SPLINE
SPL {X  -111.648, Y  +797.871, Z    +0.000, E1   -60.847, E3 +126698.241}
SPL {X  -149.288, Y  +747.285, Z    +0.000, E1   -46.770, E3 +126694.232}
SPL {X  -159.627, Y  +719.761, Z    +0.000, E1   -35.247, E3 +126699.297}
SPL {X  -164.185, Y  +697.485, Z    +0.000, E1   -20.950, E3 +126699.616}
SPL {X  -165.453, Y  +683.578, Z    +0.000, E1    -9.445, E3 +126698.203}
SPL {X  -165.642, Y  +677.105, Z    +0.000, E1    -3.559, E3 +126698.514}
SPL {X  -165.650, Y  +673.522, Z    +0.000, E1    -0.038, E3 +126697.362}
SPL {X  -165.650, Y  +671.354, Z    +0.000, E1    +3.728, E3 +126696.849}
SPL {X  -165.650, Y  +666.485, Z    +0.000, E1   +14.169, E3 +126696.576}
SPL {X  -165.650, Y  +661.236, Z    +0.000, E1   +26.072, E3 +126696.266}
SPL {X  -165.650, Y  +655.357, Z    +0.000, E1   +38.693, E3 +126695.493}
SPL {X  -165.650, Y  +646.637, Z    +0.000, E1   +52.169, E3 +126695.275}
SPL {X  -165.650, Y  +637.909, Z    +0.000, E1   +64.161, E3 +126692.070}
SPL {X  -165.650, Y  +618.963, Z    +0.000, E1   +72.815, E3 +126693.133}
SPL {X  -165.650, Y  +575.208, Z    +0.000, E1   +76.222, E3 +126704.394}
SPL {X  -165.650, Y  +394.754, Z    +0.000, E1   +73.248, E3 +126799.541}
ENDSPLINE

SPLINE
SPL {X  -165.650, Y  +407.500, Z    +0.000, E1   +70.919, E3 +126814.162}
ENDSPLINE

SPLINE
SPL {X  -165.650, Y  +384.687, Z    +0.000, E1   +71.028, E3 +126829.408}
SPL {X  -164.996, Y  +363.797, Z    +0.000, E1   +70.987, E3 +126844.383}
SPL {X  -162.841, Y  +348.123, Z    +0.000, E1   +70.683, E3 +126858.311}
SPL {X  -162.352, Y  +345.609, Z    +0.000, E1   +69.290, E3 +126872.264}
SPL {X  -157.663, Y  +327.685, Z    +0.000, E1   +69.808, E3 +126881.124}
SPL {X  -152.892, Y  +314.750, Z    +0.000, E1   +69.675, E3 +126891.339}
SPL {X  -149.246, Y  +306.628, Z    +0.000, E1   +69.029, E3 +126901.808}
SPL {X  -145.495, Y  +299.310, Z    +0.000, E1   +68.659, E3 +126909.416}
SPL {X  -142.111, Y  +293.387, Z    +0.000, E1   +68.421, E3 +126915.058}
SPL {X  -138.525, Y  +287.667, Z    +0.000, E1   +67.662, E3 +126923.618}
SPL {X  -134.450, Y  +281.737, Z    +0.000, E1   +67.268, E3 +126929.723}
SPL {X  -131.812, Y  +278.173, Z    +0.000, E1   +66.669, E3 +126935.071}
SPL {X  -128.148, Y  +273.533, Z    +0.000, E1   +67.328, E3 +126935.430}
SPL {X  -116.216, Y  +260.459, Z    +0.000, E1   +70.200, E3 +126931.736}
SPL {X   -66.125, Y  +226.621, Z    +0.000, E1   +55.862, E3 +127094.634}
ENDSPLINE

SPLINE
SPL {X  -111.531, Y  +256.023, Z    +0.000, E1   +58.853, E3 +127237.516}
SPL {X  -139.240, Y  +288.767, Z    +0.000, E1   +52.898, E3 +127247.689}
SPL {X  -156.827, Y  +325.161, Z    +0.000, E1   +39.042, E3 +127246.059}
SPL {X  -162.324, Y  +345.471, Z    +0.000, E1   +27.849, E3 +127246.527}
SPL {X  -164.696, Y  +360.744, Z    +0.000, E1   +17.229, E3 +127247.441}
SPL {X  -165.561, Y  +373.081, Z    +0.000, E1    +6.973, E3 +127246.185}
SPL {X  -165.650, Y  +379.105, Z    +0.000, E1    +1.379, E3 +127245.746}
SPL {X  -165.650, Y  +380.899, Z    +0.000, E1    -0.394, E3 +127244.884}
SPL {X  -165.650, Y  +385.044, Z    +0.000, E1    -8.496, E3 +127244.300}
SPL {X  -165.650, Y  +388.717, Z    +0.000, E1   -16.400, E3 +127244.156}
SPL {X  -165.650, Y  +394.613, Z    +0.000, E1   -29.184, E3 +127243.625}
SPL {X  -165.650, Y  +402.836, Z    +0.000, E1   -44.797, E3 +127243.027}
SPL {X  -165.650, Y  +416.111, Z    +0.000, E1   -60.729, E3 +127242.094}
SPL {X  -165.650, Y  +457.077, Z    +0.000, E1   -75.210, E3 +127245.418}
SPL {X  -165.650, Y  +475.293, Z    +0.000, E1   -75.741, E3 +127251.195}
SPL {X  -164.204, Y  +697.342, Z    +0.000, E1   -76.015, E3 +127338.170}
ENDSPLINE

SPLINE
SPL {X  -165.650, Y  +664.340, Z    +0.000, E1   -71.862, E3 +127363.574}
ENDSPLINE

SPLINE
SPL {X  -165.237, Y  +687.187, Z    +0.000, E1   -71.947, E3 +127377.835}
SPL {X  -163.865, Y  +699.752, Z    +0.000, E1   -71.643, E3 +127389.241}
SPL {X  -161.821, Y  +710.908, Z    +0.000, E1   -71.322, E3 +127399.781}
SPL {X  -158.993, Y  +721.987, Z    +0.000, E1   -71.173, E3 +127408.569}
SPL {X  -155.811, Y  +731.738, Z    +0.000, E1   -70.890, E3 +127417.577}
SPL {X  -152.643, Y  +739.844, Z    +0.000, E1   -70.463, E3 +127426.436}
SPL {X  -149.782, Y  +746.247, Z    +0.000, E1   -70.149, E3 +127433.126}
SPL {X  -146.450, Y  +752.910, Z    +0.000, E1   -69.680, E3 +127441.004}
SPL {X  -143.017, Y  +759.082, Z    +0.000, E1   -69.156, E3 +127448.615}
SPL {X  -140.057, Y  +763.953, Z    +0.000, E1   -68.829, E3 +127453.855}
SPL {X  -136.535, Y  +769.298, Z    +0.000, E1   -68.442, E3 +127459.716}
SPL {X  -133.553, Y  +773.498, Z    +0.000, E1   -67.773, E3 +127465.881}
SPL {X  -129.830, Y  +778.379, Z    +0.000, E1   -67.491, E3 +127470.507}
SPL {X  -116.788, Y  +792.975, Z    +0.000, E1   -71.297, E3 +127463.891}
SPL {X   -64.927, Y  +827.895, Z    +0.000, E1   -57.691, E3 +127589.494}
ENDSPLINE

SPLINE
SPL {X  -111.648, Y  +797.871, Z    +0.000, E1   -60.847, E3 +127786.477}
SPL {X  -149.288, Y  +747.285, Z    +0.000, E1   -46.770, E3 +127782.468}
SPL {X  -159.627, Y  +719.761, Z    +0.000, E1   -35.247, E3 +127787.533}
SPL {X  -164.185, Y  +697.485, Z    +0.000, E1   -20.950, E3 +127787.852}
SPL {X  -165.594, Y  +679.817, Z    +0.000, E1    -6.204, E3 +127786.628}
SPL {X  -165.650, Y  +673.522, Z    +0.000, E1    -0.038, E3 +127785.597}
SPL {X  -165.650, Y  +671.354, Z    +0.000, E1    +3.728, E3 +127785.085}
SPL {X  -165.650, Y  +666.485, Z    +0.000, E1   +14.169, E3 +127784.812}
SPL {X  -165.650, Y  +661.236, Z    +0.000, E1   +26.072, E3 +127784.501}
SPL {X  -165.650, Y  +655.357, Z    +0.000, E1   +38.693, E3 +127783.728}
SPL {X  -165.650, Y  +646.637, Z    +0.000, E1   +52.169, E3 +127783.510}
SPL {X  -165.650, Y  +637.909, Z    +0.000, E1   +64.161, E3 +127780.306}
SPL {X  -165.650, Y  +618.963, Z    +0.000, E1   +72.815, E3 +127781.369}
SPL {X  -165.650, Y  +575.208, Z    +0.000, E1   +76.222, E3 +127792.629}
SPL {X  -165.650, Y  +394.754, Z    +0.000, E1   +73.248, E3 +127887.776}
ENDSPLINE

SPLINE
SPL {X  -165.650, Y  +407.500, Z    +0.000, E1   +70.919, E3 +127902.397}
ENDSPLINE

SPLINE
SPL {X  -165.650, Y  +390.855, Z    +0.000, E1   +71.004, E3 +127913.325}
SPL {X  -165.534, Y  +372.295, Z    +0.000, E1   +71.066, E3 +127925.875}
SPL {X  -164.039, Y  +355.451, Z    +0.000, E1   +70.703, E3 +127941.273}
SPL {X  -161.297, Y  +340.777, Z    +0.000, E1   +70.794, E3 +127950.566}
ENDSPLINE

SPLINE
SPL {X  -162.352, Y  +345.609, Z    +0.000, E1   +69.290, E3 +127960.499}
ENDSPLINE

SPLINE
SPL {X  -159.253, Y  +332.909, Z    +0.000, E1   +69.652, E3 +127966.845}
SPL {X  -155.267, Y  +320.775, Z    +0.000, E1   +69.854, E3 +127973.939}
SPL {X  -151.256, Y  +310.961, Z    +0.000, E1   +69.467, E3 +127983.814}
SPL {X  -148.628, Y  +305.359, Z    +0.000, E1   +68.848, E3 +127992.092}
SPL {X  -145.495, Y  +299.310, Z    +0.000, E1   +68.659, E3 +127997.651}
SPL {X  -142.111, Y  +293.387, Z    +0.000, E1   +68.421, E3 +128003.293}
SPL {X  -138.525, Y  +287.667, Z    +0.000, E1   +67.662, E3 +128011.853}
SPL {X  -134.450, Y  +281.737, Z    +0.000, E1   +67.268, E3 +128017.958}
SPL {X  -131.812, Y  +278.173, Z    +0.000, E1   +66.669, E3 +128023.307}
SPL {X  -128.148, Y  +273.533, Z    +0.000, E1   +67.328, E3 +128023.665}
SPL {X  -116.216, Y  +260.459, Z    +0.000, E1   +70.200, E3 +128019.972}
SPL {X   -66.125, Y  +226.621, Z    +0.000, E1   +55.862, E3 +128182.870}
ENDSPLINE

SPLINE
SPL {X  -111.531, Y  +256.023, Z    +0.000, E1   +58.853, E3 +128325.752}
SPL {X  -139.240, Y  +288.767, Z    +0.000, E1   +52.898, E3 +128335.925}
SPL {X  -156.827, Y  +325.161, Z    +0.000, E1   +39.042, E3 +128334.294}
SPL {X  -163.133, Y  +349.734, Z    +0.000, E1   +25.193, E3 +128335.419}
SPL {X  -165.214, Y  +366.494, Z    +0.000, E1   +12.605, E3 +128334.891}
SPL {X  -165.615, Y  +375.073, Z    +0.000, E1    +5.133, E3 +128334.379}
SPL {X  -165.650, Y  +380.392, Z    +0.000, E1    +0.180, E3 +128333.338}
SPL {X  -165.650, Y  +381.828, Z    +0.000, E1    -2.219, E3 +128332.736}
SPL {X  -165.650, Y  +385.044, Z    +0.000, E1    -8.496, E3 +128332.535}
SPL {X  -165.650, Y  +388.717, Z    +0.000, E1   -16.400, E3 +128332.391}
SPL {X  -165.650, Y  +394.613, Z    +0.000, E1   -29.184, E3 +128331.860}
SPL {X  -165.650, Y  +402.836, Z    +0.000, E1   -44.797, E3 +128331.263}
SPL {X  -165.650, Y  +416.111, Z    +0.000, E1   -60.729, E3 +128330.329}
SPL {X  -165.650, Y  +471.994, Z    +0.000, E1   -75.670, E3 +128338.383}
SPL {X  -164.204, Y  +697.342, Z    +0.000, E1   -76.015, E3 +128426.405}
ENDSPLINE

SPLINE
SPL {X  -165.650, Y  +664.340, Z    +0.000, E1   -71.862, E3 +128451.809}
ENDSPLINE

SPLINE
SPL {X  -165.237, Y  +687.187, Z    +0.000, E1   -71.947, E3 +128466.070}
SPL {X  -163.865, Y  +699.752, Z    +0.000, E1   -71.643, E3 +128477.476}
SPL {X  -161.821, Y  +710.908, Z    +0.000, E1   -71.322, E3 +128488.016}
SPL {X  -158.993, Y  +721.987, Z    +0.000, E1   -71.173, E3 +128496.804}
SPL {X  -155.811, Y  +731.738, Z    +0.000, E1   -70.890, E3 +128505.812}
SPL {X  -152.643, Y  +739.844, Z    +0.000, E1   -70.463, E3 +128514.672}
SPL {X  -149.782, Y  +746.247, Z    +0.000, E1   -70.149, E3 +128521.361}
SPL {X  -146.450, Y  +752.910, Z    +0.000, E1   -69.680, E3 +128529.239}
SPL {X  -143.017, Y  +759.082, Z    +0.000, E1   -69.156, E3 +128536.851}
SPL {X  -140.057, Y  +763.953, Z    +0.000, E1   -68.829, E3 +128542.090}
SPL {X  -136.535, Y  +769.298, Z    +0.000, E1   -68.442, E3 +128547.952}
SPL {X  -132.359, Y  +775.105, Z    +0.000, E1   -67.661, E3 +128555.809}
SPL {X  -128.720, Y  +779.765, Z    +0.000, E1   -67.454, E3 +128559.790}
SPL {X  -116.788, Y  +792.975, Z    +0.000, E1   -71.297, E3 +128552.127}
SPL {X   -70.520, Y  +825.390, Z    +0.000, E1   -59.928, E3 +128646.037}
SPL {X   -62.607, Y  +828.863, Z    +0.000, E1   -56.584, E3 +128700.922}
ENDSPLINE

SPLINE
SPL {X  -111.648, Y  +797.871, Z    +0.000, E1   -60.847, E3 +128874.712}
SPL {X  -149.288, Y  +747.285, Z    +0.000, E1   -46.770, E3 +128870.703}
SPL {X  -161.496, Y  +712.364, Z    +0.000, E1   -31.137, E3 +128876.498}
SPL {X  -164.701, Y  +693.202, Z    +0.000, E1   -17.512, E3 +128875.472}
SPL {X  -165.594, Y  +679.817, Z    +0.000, E1    -6.204, E3 +128874.863}
SPL {X  -165.650, Y  +673.263, Z    +0.000, E1    +0.216, E3 +128873.745}
SPL {X  -165.650, Y  +670.095, Z    +0.000, E1    +6.482, E3 +128873.148}
SPL {X  -165.650, Y  +666.485, Z    +0.000, E1   +14.169, E3 +128873.047}
SPL {X  -165.650, Y  +661.236, Z    +0.000, E1   +26.072, E3 +128872.736}
SPL {X  -165.650, Y  +655.357, Z    +0.000, E1   +38.693, E3 +128871.964}
SPL {X  -165.650, Y  +646.637, Z    +0.000, E1   +52.169, E3 +128871.745}
SPL {X  -165.650, Y  +637.909, Z    +0.000, E1   +64.161, E3 +128868.541}
SPL {X  -165.650, Y  +618.963, Z    +0.000, E1   +72.815, E3 +128869.604}
SPL {X  -165.650, Y  +575.208, Z    +0.000, E1   +76.222, E3 +128880.865}
SPL {X  -165.650, Y  +394.754, Z    +0.000, E1   +73.248, E3 +128976.011}
ENDSPLINE

SPLINE
SPL {X  -165.650, Y  +407.500, Z    +0.000, E1   +70.919, E3 +128990.632}
ENDSPLINE

SPLINE
SPL {X  -165.650, Y  +390.855, Z    +0.000, E1   +71.004, E3 +129001.560}
SPL {X  -165.534, Y  +372.295, Z    +0.000, E1   +71.066, E3 +129014.110}
SPL {X  -164.039, Y  +355.451, Z    +0.000, E1   +70.703, E3 +129029.509}
SPL {X  -161.297, Y  +340.777, Z    +0.000, E1   +70.794, E3 +129038.801}
ENDSPLINE

SPLINE
SPL {X  -162.352, Y  +345.609, Z    +0.000, E1   +69.290, E3 +129048.734}
ENDSPLINE

SPLINE
SPL {X  -157.663, Y  +327.685, Z    +0.000, E1   +69.808, E3 +129057.594}
SPL {X  -152.892, Y  +314.750, Z    +0.000, E1   +69.675, E3 +129067.810}
SPL {X  -149.246, Y  +306.628, Z    +0.000, E1   +69.029, E3 +129078.278}
SPL {X  -145.495, Y  +299.310, Z    +0.000, E1   +68.659, E3 +129085.887}
SPL {X  -142.111, Y  +293.387, Z    +0.000, E1   +68.421, E3 +129091.528}
SPL {X  -138.525, Y  +287.667, Z    +0.000, E1   +67.662, E3 +129100.088}
SPL {X  -134.450, Y  +281.737, Z    +0.000, E1   +67.268, E3 +129106.193}
SPL {X  -131.812, Y  +278.173, Z    +0.000, E1   +66.669, E3 +129111.542}
SPL {X  -128.148, Y  +273.533, Z    +0.000, E1   +67.328, E3 +129111.900}
SPL {X  -116.216, Y  +260.459, Z    +0.000, E1   +70.200, E3 +129108.207}
SPL {X   -66.125, Y  +226.621, Z    +0.000, E1   +55.862, E3 +129271.105}
ENDSPLINE

SPLINE
SPL {X  -111.531, Y  +256.023, Z    +0.000, E1   +58.853, E3 +129413.987}
SPL {X  -139.240, Y  +288.767, Z    +0.000, E1   +52.898, E3 +129424.160}
SPL {X  -156.827, Y  +325.161, Z    +0.000, E1   +39.042, E3 +129422.529}
SPL {X  -162.324, Y  +345.471, Z    +0.000, E1   +27.849, E3 +129422.998}
SPL {X  -165.055, Y  +364.477, Z    +0.000, E1   +14.326, E3 +129423.436}
SPL {X  -165.646, Y  +377.353, Z    +0.000, E1    +3.112, E3 +129422.393}
SPL {X  -165.650, Y  +380.500, Z    +0.000, E1    -0.000, E3 +129421.519}
SPL {X  -165.650, Y  +381.828, Z    +0.000, E1    -2.219, E3 +129420.971}
SPL {X  -165.650, Y  +385.044, Z    +0.000, E1    -8.496, E3 +129420.771}
SPL {X  -165.650, Y  +390.492, Z    +0.000, E1   -20.084, E3 +129420.425}
SPL {X  -165.650, Y  +400.081, Z    +0.000, E1   -39.836, E3 +129419.730}
SPL {X  -165.650, Y  +416.111, Z    +0.000, E1   -60.729, E3 +129418.565}
SPL {X  -165.650, Y  +471.994, Z    +0.000, E1   -75.670, E3 +129426.618}
SPL {X  -164.204, Y  +697.342, Z    +0.000, E1   -76.015, E3 +129514.641}
ENDSPLINE

SPLINE
SPL {X  -165.650, Y  +656.030, Z    +0.000, E1   -71.686, E3 +129536.080}
ENDSPLINE

SPLINE
SPL {X  -165.610, Y  +679.119, Z    +0.000, E1   -71.889, E3 +129549.703}
SPL {X  -163.827, Y  +700.009, Z    +0.000, E1   -71.824, E3 +129564.269}
SPL {X  -161.041, Y  +714.304, Z    +0.000, E1   -71.423, E3 +129577.615}
SPL {X  -159.124, Y  +721.538, Z    +0.000, E1   -70.872, E3 +129587.267}
SPL {X  -155.811, Y  +731.738, Z    +0.000, E1   -70.890, E3 +129594.048}
SPL {X  -152.643, Y  +739.844, Z    +0.000, E1   -70.463, E3 +129602.907}
SPL {X  -149.782, Y  +746.247, Z    +0.000, E1   -70.149, E3 +129609.597}
SPL {X  -146.450, Y  +752.910, Z    +0.000, E1   -69.680, E3 +129617.475}
SPL {X  -143.017, Y  +759.082, Z    +0.000, E1   -69.156, E3 +129625.086}
SPL {X  -139.030, Y  +765.558, Z    +0.000, E1   -68.719, E3 +129632.119}
SPL {X  -135.682, Y  +770.527, Z    +0.000, E1   -68.337, E3 +129637.503}
SPL {X  -133.553, Y  +773.498, Z    +0.000, E1   -67.773, E3 +129642.352}
SPL {X  -129.830, Y  +778.379, Z    +0.000, E1   -67.491, E3 +129646.978}
SPL {X  -116.788, Y  +792.975, Z    +0.000, E1   -71.297, E3 +129640.362}
SPL {X   -70.520, Y  +825.390, Z    +0.000, E1   -59.928, E3 +129734.272}
SPL {X   -62.607, Y  +828.863, Z    +0.000, E1   -56.584, E3 +129789.157}
ENDSPLINE

SPLINE
SPL {X  -111.648, Y  +797.871, Z    +0.000, E1   -60.847, E3 +129962.947}
SPL {X  -149.288, Y  +747.285, Z    +0.000, E1   -46.770, E3 +129958.938}
SPL {X  -161.496, Y  +712.364, Z    +0.000, E1   -31.137, E3 +129964.733}
SPL {X  -164.701, Y  +693.202, Z    +0.000, E1   -17.512, E3 +129963.708}
SPL {X  -165.453, Y  +683.578, Z    +0.000, E1    -9.445, E3 +129962.909}
SPL {X  -165.642, Y  +677.105, Z    +0.000, E1    -3.559, E3 +129963.220}
SPL {X  -165.650, Y  +673.263, Z    +0.000, E1    +0.216, E3 +129961.980}
SPL {X  -165.650, Y  +670.095, Z    +0.000, E1    +6.482, E3 +129961.384}
SPL {X  -165.650, Y  +666.485, Z    +0.000, E1   +14.169, E3 +129961.282}
SPL {X  -165.650, Y  +661.236, Z    +0.000, E1   +26.072, E3 +129960.971}
SPL {X  -165.650, Y  +653.063, Z    +0.000, E1   +42.395, E3 +129960.375}
SPL {X  -165.650, Y  +640.535, Z    +0.000, E1   +60.776, E3 +129957.860}
SPL {X  -165.650, Y  +618.963, Z    +0.000, E1   +72.815, E3 +129957.839}
SPL {X  -165.650, Y  +575.208, Z    +0.000, E1   +76.222, E3 +129969.100}
SPL {X  -165.650, Y  +394.754, Z    +0.000, E1   +73.248, E3 +130064.246}
ENDSPLINE

SPLINE
SPL {X  -165.650, Y  +407.500, Z    +0.000, E1   +70.919, E3 +130078.868}
ENDSPLINE

SPLINE
SPL {X  -165.650, Y  +384.687, Z    +0.000, E1   +71.028, E3 +130094.114}
SPL {X  -164.996, Y  +363.797, Z    +0.000, E1   +70.987, E3 +130109.089}
SPL {X  -162.841, Y  +348.123, Z    +0.000, E1   +70.683, E3 +130123.016}
SPL {X  -162.352, Y  +345.609, Z    +0.000, E1   +69.290, E3 +130136.969}
SPL {X  -159.253, Y  +332.909, Z    +0.000, E1   +69.652, E3 +130143.316}
SPL {X  -156.309, Y  +323.661, Z    +0.000, E1   +69.908, E3 +130147.831}
SPL {X  -152.892, Y  +314.750, Z    +0.000, E1   +69.675, E3 +130156.045}
SPL {X  -149.246, Y  +306.628, Z    +0.000, E1   +69.029, E3 +130166.513}
SPL {X  -144.614, Y  +297.712, Z    +0.000, E1   +68.717, E3 +130174.867}
SPL {X  -141.011, Y  +291.576, Z    +0.000, E1   +68.040, E3 +130183.345}
SPL {X  -137.649, Y  +286.345, Z    +0.000, E1   +67.498, E3 +130190.039}
SPL {X  -134.450, Y  +281.737, Z    +0.000, E1   +67.268, E3 +130194.429}
SPL {X  -131.812, Y  +278.173, Z    +0.000, E1   +66.669, E3 +130199.777}
SPL {X  -128.148, Y  +273.533, Z    +0.000, E1   +67.328, E3 +130200.136}
SPL {X  -116.216, Y  +260.459, Z    +0.000, E1   +70.200, E3 +130196.442}
SPL {X   -66.125, Y  +226.621, Z    +0.000, E1   +55.862, E3 +130359.340}
ENDSPLINE

SPLINE
SPL {X  -111.531, Y  +256.023, Z    +0.000, E1   +58.853, E3 +130502.222}
SPL {X  -139.240, Y  +288.767, Z    +0.000, E1   +52.898, E3 +130512.395}
SPL {X  -156.827, Y  +325.161, Z    +0.000, E1   +39.042, E3 +130510.764}
SPL {X  -162.324, Y  +345.471, Z    +0.000, E1   +27.849, E3 +130511.233}
SPL {X  -164.696, Y  +360.744, Z    +0.000, E1   +17.229, E3 +130512.147}
SPL {X  -165.561, Y  +373.081, Z    +0.000, E1    +6.973, E3 +130510.891}
SPL {X  -165.650, Y  +379.105, Z    +0.000, E1    +1.379, E3 +130510.452}
SPL {X  -165.650, Y  +380.899, Z    +0.000, E1    -0.394, E3 +130509.590}
SPL {X  -165.650, Y  +385.044, Z    +0.000, E1    -8.496, E3 +130509.006}
SPL {X  -165.650, Y  +388.717, Z    +0.000, E1   -16.400, E3 +130508.862}
SPL {X  -165.650, Y  +394.613, Z    +0.000, E1   -29.184, E3 +130508.331}
SPL {X  -165.650, Y  +402.836, Z    +0.000, E1   -44.797, E3 +130507.733}
SPL {X  -165.650, Y  +416.111, Z    +0.000, E1   -60.729, E3 +130506.800}
SPL {X  -165.650, Y  +457.077, Z    +0.000, E1   -75.210, E3 +130510.123}
SPL {X  -165.650, Y  +475.293, Z    +0.000, E1   -75.741, E3 +130515.901}
SPL {X  -164.204, Y  +697.342, Z    +0.000, E1   -76.015, E3 +130602.876}
ENDSPLINE

SPLINE
SPL {X  -165.650, Y  +664.340, Z    +0.000, E1   -71.862, E3 +130628.279}
ENDSPLINE

SPLINE
SPL {X  -165.237, Y  +687.187, Z    +0.000, E1   -71.947, E3 +130642.541}
SPL {X  -163.865, Y  +699.752, Z    +0.000, E1   -71.643, E3 +130653.947}
SPL {X  -161.821, Y  +710.908, Z    +0.000, E1   -71.322, E3 +130664.487}
SPL {X  -158.993, Y  +721.987, Z    +0.000, E1   -71.173, E3 +130673.275}
SPL {X  -155.811, Y  +731.738, Z    +0.000, E1   -70.890, E3 +130682.283}
SPL {X  -152.643, Y  +739.844, Z    +0.000, E1   -70.463, E3 +130691.142}
SPL {X  -149.782, Y  +746.247, Z    +0.000, E1   -70.149, E3 +130697.832}
SPL {X  -146.450, Y  +752.910, Z    +0.000, E1   -69.680, E3 +130705.710}
SPL {X  -143.017, Y  +759.082, Z    +0.000, E1   -69.156, E3 +130713.321}
SPL {X  -140.057, Y  +763.953, Z    +0.000, E1   -68.829, E3 +130718.561}
SPL {X  -136.535, Y  +769.298, Z    +0.000, E1   -68.442, E3 +130724.422}
SPL {X  -133.553, Y  +773.498, Z    +0.000, E1   -67.773, E3 +130730.587}
SPL {X  -129.830, Y  +778.379, Z    +0.000, E1   -67.491, E3 +130735.213}
SPL {X  -116.788, Y  +792.975, Z    +0.000, E1   -71.297, E3 +130728.597}
SPL {X   -64.927, Y  +827.895, Z    +0.000, E1   -57.691, E3 +130854.200}
ENDSPLINE

SPLINE
SPL {X  -111.648, Y  +797.871, Z    +0.000, E1   -60.847, E3 +131051.183}
SPL {X  -149.288, Y  +747.285, Z    +0.000, E1   -46.770, E3 +131047.173}
SPL {X  -159.627, Y  +719.761, Z    +0.000, E1   -35.247, E3 +131052.239}
SPL {X  -164.185, Y  +697.485, Z    +0.000, E1   -20.950, E3 +131052.557}
SPL {X  -165.594, Y  +679.817, Z    +0.000, E1    -6.204, E3 +131051.334}
SPL {X  -165.650, Y  +673.522, Z    +0.000, E1    -0.038, E3 +131050.303}
SPL {X  -165.650, Y  +671.354, Z    +0.000, E1    +3.728, E3 +131049.790}
SPL {X  -165.650, Y  +666.485, Z    +0.000, E1   +14.169, E3 +131049.518}
SPL {X  -165.650, Y  +661.236, Z    +0.000, E1   +26.072, E3 +131049.207}
SPL {X  -165.650, Y  +655.357, Z    +0.000, E1   +38.693, E3 +131048.434}
SPL {X  -165.650, Y  +646.637, Z    +0.000, E1   +52.169, E3 +131048.216}
SPL {X  -165.650, Y  +637.909, Z    +0.000, E1   +64.161, E3 +131045.011}
SPL {X  -165.650, Y  +618.963, Z    +0.000, E1   +72.815, E3 +131046.075}
SPL {X  -165.650, Y  +575.208, Z    +0.000, E1   +76.222, E3 +131057.335}
SPL {X  -165.650, Y  +394.754, Z    +0.000, E1   +73.248, E3 +131152.482}
ENDSPLINE

SPLINE
SPL {X  -165.650, Y  +407.500, Z    +0.000, E1   +70.919, E3 +131167.103}
ENDSPLINE

SPLINE
SPL {X  -165.650, Y  +390.855, Z    +0.000, E1   +71.004, E3 +131178.031}
SPL {X  -165.534, Y  +372.295, Z    +0.000, E1   +71.066, E3 +131190.581}
SPL {X  -164.039, Y  +355.451, Z    +0.000, E1   +70.703, E3 +131205.979}
SPL {X  -161.297, Y  +340.777, Z    +0.000, E1   +70.794, E3 +131215.272}
ENDSPLINE

SPLINE
SPL {X  -162.352, Y  +345.609, Z    +0.000, E1   +69.290, E3 +131225.205}
ENDSPLINE

SPLINE
SPL {X  -159.253, Y  +332.909, Z    +0.000, E1   +69.652, E3 +131231.551}
SPL {X  -155.267, Y  +320.775, Z    +0.000, E1   +69.854, E3 +131238.645}
SPL {X  -151.256, Y  +310.961, Z    +0.000, E1   +69.467, E3 +131248.519}
SPL {X  -148.628, Y  +305.359, Z    +0.000, E1   +68.848, E3 +131256.798}
SPL {X  -145.495, Y  +299.310, Z    +0.000, E1   +68.659, E3 +131262.357}
SPL {X  -142.111, Y  +293.387, Z    +0.000, E1   +68.421, E3 +131267.999}
SPL {X  -138.525, Y  +287.667, Z    +0.000, E1   +67.662, E3 +131276.559}
SPL {X  -134.450, Y  +281.737, Z    +0.000, E1   +67.268, E3 +131282.664}
SPL {X  -131.812, Y  +278.173, Z    +0.000, E1   +66.669, E3 +131288.012}
SPL {X  -128.148, Y  +273.533, Z    +0.000, E1   +67.328, E3 +131288.371}
SPL {X  -116.216, Y  +260.459, Z    +0.000, E1   +70.200, E3 +131284.677}
SPL {X   -66.125, Y  +226.621, Z    +0.000, E1   +55.862, E3 +131447.576}
ENDSPLINE

SPLINE
SPL {X  -111.531, Y  +256.023, Z    +0.000, E1   +58.853, E3 +131590.458}
SPL {X  -139.240, Y  +288.767, Z    +0.000, E1   +52.898, E3 +131600.630}
SPL {X  -156.827, Y  +325.161, Z    +0.000, E1   +39.042, E3 +131599.000}
SPL {X  -163.133, Y  +349.734, Z    +0.000, E1   +25.193, E3 +131600.124}
SPL {X  -165.214, Y  +366.494, Z    +0.000, E1   +12.605, E3 +131599.597}
SPL {X  -165.615, Y  +375.073, Z    +0.000, E1    +5.133, E3 +131599.085}
SPL {X  -165.650, Y  +380.392, Z    +0.000, E1    +0.180, E3 +131598.044}
SPL {X  -165.650, Y  +381.828, Z    +0.000, E1    -2.219, E3 +131597.442}
SPL {X  -165.650, Y  +385.044, Z    +0.000, E1    -8.496, E3 +131597.241}
SPL {X  -165.650, Y  +388.717, Z    +0.000, E1   -16.400, E3 +131597.097}
SPL {X  -165.650, Y  +394.613, Z    +0.000, E1   -29.184, E3 +131596.566}
SPL {X  -165.650, Y  +402.836, Z    +0.000, E1   -44.797, E3 +131595.969}
SPL {X  -165.650, Y  +416.111, Z    +0.000, E1   -60.729, E3 +131595.035}
SPL {X  -165.650, Y  +471.994, Z    +0.000, E1   -75.670, E3 +131603.088}
SPL {X  -164.204, Y  +697.342, Z    +0.000, E1   -76.015, E3 +131691.111}
ENDSPLINE

SPLINE
SPL {X  -165.650, Y  +656.030, Z    +0.000, E1   -71.686, E3 +131712.551}
ENDSPLINE

SPLINE
SPL {X  -165.610, Y  +679.119, Z    +0.000, E1   -71.889, E3 +131726.174}
SPL {X  -163.827, Y  +700.009, Z    +0.000, E1   -71.824, E3 +131740.740}
SPL {X  -161.821, Y  +710.908, Z    +0.000, E1   -71.322, E3 +131752.722}
SPL {X  -158.993, Y  +721.987, Z    +0.000, E1   -71.173, E3 +131761.510}
SPL {X  -155.811, Y  +731.738, Z    +0.000, E1   -70.890, E3 +131770.518}
SPL {X  -152.643, Y  +739.844, Z    +0.000, E1   -70.463, E3 +131779.377}
SPL {X  -149.782, Y  +746.247, Z    +0.000, E1   -70.149, E3 +131786.067}
SPL {X  -146.450, Y  +752.910, Z    +0.000, E1   -69.680, E3 +131793.945}
SPL {X  -143.017, Y  +759.082, Z    +0.000, E1   -69.156, E3 +131801.557}
SPL {X  -140.057, Y  +763.953, Z    +0.000, E1   -68.829, E3 +131806.796}
SPL {X  -136.535, Y  +769.298, Z    +0.000, E1   -68.442, E3 +131812.658}
SPL {X  -132.359, Y  +775.105, Z    +0.000, E1   -67.661, E3 +131820.515}
SPL {X  -128.720, Y  +779.765, Z    +0.000, E1   -67.454, E3 +131824.496}
SPL {X  -116.788, Y  +792.975, Z    +0.000, E1   -71.297, E3 +131816.833}
SPL {X   -64.927, Y  +827.895, Z    +0.000, E1   -57.691, E3 +131942.435}
ENDSPLINE

SPLINE
SPL {X  -111.648, Y  +797.871, Z    +0.000, E1   -60.847, E3 +132139.418}
SPL {X  -149.288, Y  +747.285, Z    +0.000, E1   -46.770, E3 +132135.409}
SPL {X  -159.627, Y  +719.761, Z    +0.000, E1   -35.247, E3 +132140.474}
SPL {X  -164.185, Y  +697.485, Z    +0.000, E1   -20.950, E3 +132140.793}
SPL {X  -165.594, Y  +679.817, Z    +0.000, E1    -6.204, E3 +132139.569}
SPL {X  -165.650, Y  +673.522, Z    +0.000, E1    -0.038, E3 +132138.538}
SPL {X  -165.650, Y  +671.354, Z    +0.000, E1    +3.728, E3 +132138.026}
SPL {X  -165.650, Y  +666.485, Z    +0.000, E1   +14.169, E3 +132137.753}
SPL {X  -165.650, Y  +661.236, Z    +0.000, E1   +26.072, E3 +132137.442}
SPL {X  -165.650, Y  +655.357, Z    +0.000, E1   +38.693, E3 +132136.670}
SPL {X  -165.650, Y  +646.637, Z    +0.000, E1   +52.169, E3 +132136.451}
SPL {X  -165.650, Y  +637.909, Z    +0.000, E1   +64.161, E3 +132133.247}
SPL {X  -165.650, Y  +618.963, Z    +0.000, E1   +72.815, E3 +132134.310}
SPL {X  -165.650, Y  +582.897, Z    +0.000, E1   +76.147, E3 +132142.971}
SPL {X  -165.650, Y  +558.388, Z    +0.000, E1   +76.294, E3 +132151.283}
SPL {X  -165.650, Y  +391.690, Z    +0.000, E1   +75.504, E3 +132221.050}
ENDSPLINE

SPLINE
SPL {X  -165.650, Y  +396.283, Z    +0.000, E1   +72.775, E3 +132244.355}
SPL {X  -165.650, Y  +407.500, Z    +0.000, E1   +70.919, E3 +132255.338}
ENDSPLINE

SPLINE
SPL {X  -165.650, Y  +390.855, Z    +0.000, E1   +71.004, E3 +132266.266}
SPL {X  -165.534, Y  +372.295, Z    +0.000, E1   +71.066, E3 +132278.816}
SPL {X  -164.687, Y  +360.663, Z    +0.000, E1   +70.826, E3 +132289.108}
SPL {X  -162.841, Y  +348.123, Z    +0.000, E1   +70.683, E3 +132299.487}
SPL {X  -162.352, Y  +345.609, Z    +0.000, E1   +69.290, E3 +132313.440}
SPL {X  -159.253, Y  +332.909, Z    +0.000, E1   +69.652, E3 +132319.786}
SPL {X  -156.309, Y  +323.661, Z    +0.000, E1   +69.908, E3 +132324.301}
SPL {X  -152.892, Y  +314.750, Z    +0.000, E1   +69.675, E3 +132332.516}
SPL {X  -149.246, Y  +306.628, Z    +0.000, E1   +69.029, E3 +132342.984}
SPL {X  -145.495, Y  +299.310, Z    +0.000, E1   +68.659, E3 +132350.593}
SPL {X  -142.111, Y  +293.387, Z    +0.000, E1   +68.421, E3 +132356.234}
SPL {X  -138.525, Y  +287.667, Z    +0.000, E1   +67.662, E3 +132364.794}
SPL {X  -134.450, Y  +281.737, Z    +0.000, E1   +67.268, E3 +132370.899}
SPL {X  -131.812, Y  +278.173, Z    +0.000, E1   +66.669, E3 +132376.248}
SPL {X  -128.148, Y  +273.533, Z    +0.000, E1   +67.328, E3 +132376.606}
SPL {X  -116.216, Y  +260.459, Z    +0.000, E1   +70.200, E3 +132372.913}
SPL {X   -66.125, Y  +226.621, Z    +0.000, E1   +55.862, E3 +132535.811}
ENDSPLINE

SPLINE
SPL {X  -111.531, Y  +256.023, Z    +0.000, E1   +58.853, E3 +132678.693}
SPL {X  -139.240, Y  +288.767, Z    +0.000, E1   +52.898, E3 +132688.866}
SPL {X  -156.827, Y  +325.161, Z    +0.000, E1   +39.042, E3 +132687.235}
SPL {X  -162.324, Y  +345.471, Z    +0.000, E1   +27.849, E3 +132687.704}
SPL {X  -165.055, Y  +364.477, Z    +0.000, E1   +14.326, E3 +132688.142}
SPL {X  -165.646, Y  +377.353, Z    +0.000, E1    +3.112, E3 +132687.099}
SPL {X  -165.650, Y  +380.500, Z    +0.000, E1    -0.000, E3 +132686.225}
SPL {X  -165.650, Y  +381.828, Z    +0.000, E1    -2.219, E3 +132685.677}
SPL {X  -165.650, Y  +385.044, Z    +0.000, E1    -8.496, E3 +132685.477}
SPL {X  -165.650, Y  +390.492, Z    +0.000, E1   -20.084, E3 +132685.131}
SPL {X  -165.650, Y  +400.081, Z    +0.000, E1   -39.836, E3 +132684.436}
SPL {X  -165.650, Y  +416.111, Z    +0.000, E1   -60.729, E3 +132683.270}
SPL {X  -165.650, Y  +471.994, Z    +0.000, E1   -75.670, E3 +132691.324}
SPL {X  -164.204, Y  +697.342, Z    +0.000, E1   -76.015, E3 +132779.346}
ENDSPLINE

SPLINE
SPL {X  -165.650, Y  +656.030, Z    +0.000, E1   -71.686, E3 +132800.786}
ENDSPLINE

SPLINE
SPL {X  -165.610, Y  +679.119, Z    +0.000, E1   -71.889, E3 +132814.409}
SPL {X  -163.827, Y  +700.009, Z    +0.000, E1   -71.824, E3 +132828.975}
SPL {X  -161.821, Y  +710.908, Z    +0.000, E1   -71.322, E3 +132840.957}
SPL {X  -158.993, Y  +721.987, Z    +0.000, E1   -71.173, E3 +132849.746}
SPL {X  -155.811, Y  +731.738, Z    +0.000, E1   -70.890, E3 +132858.753}
SPL {X  -152.643, Y  +739.844, Z    +0.000, E1   -70.463, E3 +132867.613}
SPL {X  -149.782, Y  +746.247, Z    +0.000, E1   -70.149, E3 +132874.302}
SPL {X  -146.450, Y  +752.910, Z    +0.000, E1   -69.680, E3 +132882.181}
SPL {X  -143.017, Y  +759.082, Z    +0.000, E1   -69.156, E3 +132889.792}
SPL {X  -140.057, Y  +763.953, Z    +0.000, E1   -68.829, E3 +132895.031}
SPL {X  -136.535, Y  +769.298, Z    +0.000, E1   -68.442, E3 +132900.893}
SPL {X  -132.359, Y  +775.105, Z    +0.000, E1   -67.661, E3 +132908.750}
SPL {X  -128.720, Y  +779.765, Z    +0.000, E1   -67.454, E3 +132912.731}
SPL {X  -116.788, Y  +792.975, Z    +0.000, E1   -71.297, E3 +132905.068}
SPL {X   -64.927, Y  +827.895, Z    +0.000, E1   -57.691, E3 +133030.671}
ENDSPLINE

SPLINE
SPL {X  -111.648, Y  +797.871, Z    +0.000, E1   -60.847, E3 +133227.653}
SPL {X  -149.288, Y  +747.285, Z    +0.000, E1   -46.770, E3 +133223.644}
SPL {X  -161.496, Y  +712.364, Z    +0.000, E1   -31.137, E3 +133229.439}
SPL {X  -164.701, Y  +693.202, Z    +0.000, E1   -17.512, E3 +133228.413}
SPL {X  -165.453, Y  +683.578, Z    +0.000, E1    -9.445, E3 +133227.615}
SPL {X  -165.642, Y  +677.105, Z    +0.000, E1    -3.559, E3 +133227.926}
SPL {X  -165.650, Y  +673.522, Z    +0.000, E1    -0.038, E3 +133226.773}
SPL {X  -165.650, Y  +671.354, Z    +0.000, E1    +3.728, E3 +133226.261}
SPL {X  -165.650, Y  +666.485, Z    +0.000, E1   +14.169, E3 +133225.988}
SPL {X  -165.650, Y  +661.236, Z    +0.000, E1   +26.072, E3 +133225.677}
SPL {X  -165.650, Y  +653.063, Z    +0.000, E1   +42.395, E3 +133225.081}
SPL {X  -165.650, Y  +640.535, Z    +0.000, E1   +60.776, E3 +133222.566}
SPL {X  -165.650, Y  +618.963, Z    +0.000, E1   +72.815, E3 +133222.545}
SPL {X  -165.650, Y  +575.208, Z    +0.000, E1   +76.222, E3 +133233.806}
SPL {X  -165.650, Y  +394.754, Z    +0.000, E1   +73.248, E3 +133328.952}
ENDSPLINE

SPLINE
SPL {X  -165.650, Y  +407.500, Z    +0.000, E1   +70.919, E3 +133343.574}
ENDSPLINE

SPLINE
SPL {X  -165.650, Y  +390.855, Z    +0.000, E1   +71.004, E3 +133354.501}
SPL {X  -165.534, Y  +372.295, Z    +0.000, E1   +71.066, E3 +133367.052}
SPL {X  -164.039, Y  +355.451, Z    +0.000, E1   +70.703, E3 +133382.450}
SPL {X  -161.297, Y  +340.777, Z    +0.000, E1   +70.794, E3 +133391.742}
ENDSPLINE

SPLINE
SPL {X  -162.352, Y  +345.609, Z    +0.000, E1   +69.290, E3 +133401.675}
ENDSPLINE

SPLINE
SPL {X  -157.663, Y  +327.685, Z    +0.000, E1   +69.808, E3 +133410.536}
SPL {X  -152.892, Y  +314.750, Z    +0.000, E1   +69.675, E3 +133420.751}
SPL {X  -149.246, Y  +306.628, Z    +0.000, E1   +69.029, E3 +133431.219}
SPL {X  -145.495, Y  +299.310, Z    +0.000, E1   +68.659, E3 +133438.828}
SPL {X  -142.111, Y  +293.387, Z    +0.000, E1   +68.421, E3 +133444.470}
SPL {X  -138.525, Y  +287.667, Z    +0.000, E1   +67.662, E3 +133453.029}
SPL {X  -134.450, Y  +281.737, Z    +0.000, E1   +67.268, E3 +133459.135}
SPL {X  -131.812, Y  +278.173, Z    +0.000, E1   +66.669, E3 +133464.483}
SPL {X  -128.148, Y  +273.533, Z    +0.000, E1   +67.328, E3 +133464.842}
SPL {X  -116.216, Y  +260.459, Z    +0.000, E1   +70.200, E3 +133461.148}
SPL {X   -66.125, Y  +226.621, Z    +0.000, E1   +55.862, E3 +133624.046}
ENDSPLINE

SPLINE
SPL {X  -111.531, Y  +256.023, Z    +0.000, E1   +58.853, E3 +133766.928}
SPL {X  -139.240, Y  +288.767, Z    +0.000, E1   +52.898, E3 +133777.101}
SPL {X  -156.827, Y  +325.161, Z    +0.000, E1   +39.042, E3 +133775.470}
SPL {X  -163.133, Y  +349.734, Z    +0.000, E1   +25.193, E3 +133776.595}
SPL {X  -165.214, Y  +366.494, Z    +0.000, E1   +12.605, E3 +133776.068}
SPL {X  -165.646, Y  +377.353, Z    +0.000, E1    +3.112, E3 +133775.334}
SPL {X  -165.650, Y  +380.899, Z    +0.000, E1    -0.394, E3 +133774.296}
SPL {X  -165.650, Y  +385.044, Z    +0.000, E1    -8.496, E3 +133773.712}
SPL {X  -165.650, Y  +388.717, Z    +0.000, E1   -16.400, E3 +133773.568}
SPL {X  -165.650, Y  +392.701, Z    +0.000, E1   -25.323, E3 +133773.115}
SPL {X  -165.650, Y  +398.793, Z    +0.000, E1   -37.509, E3 +133772.884}
SPL {X  -165.650, Y  +409.325, Z    +0.000, E1   -54.181, E3 +133771.564}
SPL {X  -165.650, Y  +420.423, Z    +0.000, E1   -63.808, E3 +133771.713}
SPL {X  -165.650, Y  +471.994, Z    +0.000, E1   -75.670, E3 +133779.559}
SPL {X  -164.204, Y  +697.342, Z    +0.000, E1   -76.015, E3 +133867.582}
ENDSPLINE

SPLINE
SPL {X  -165.650, Y  +656.030, Z    +0.000, E1   -71.686, E3 +133889.021}
ENDSPLINE

SPLINE
SPL {X  -165.610, Y  +679.119, Z    +0.000, E1   -71.889, E3 +133902.645}
SPL {X  -164.561, Y  +694.465, Z    +0.000, E1   -71.736, E3 +133914.278}
SPL {X  -162.089, Y  +709.665, Z    +0.000, E1   -71.739, E3 +133924.478}
SPL {X  -159.776, Y  +719.221, Z    +0.000, E1   -71.038, E3 +133937.301}
SPL {X  -155.811, Y  +731.738, Z    +0.000, E1   -70.890, E3 +133946.989}
SPL {X  -152.643, Y  +739.844, Z    +0.000, E1   -70.463, E3 +133955.848}
SPL {X  -149.782, Y  +746.247, Z    +0.000, E1   -70.149, E3 +133962.538}
SPL {X  -146.450, Y  +752.910, Z    +0.000, E1   -69.680, E3 +133970.416}
SPL {X  -143.017, Y  +759.082, Z    +0.000, E1   -69.156, E3 +133978.027}
SPL {X  -139.030, Y  +765.558, Z    +0.000, E1   -68.719, E3 +133985.060}
SPL {X  -134.589, Y  +772.070, Z    +0.000, E1   -68.090, E3 +133992.909}
SPL {X  -129.830, Y  +778.379, Z    +0.000, E1   -67.491, E3 +133999.919}
SPL {X  -116.788, Y  +792.975, Z    +0.000, E1   -71.297, E3 +133993.303}
SPL {X   -64.927, Y  +827.895, Z    +0.000, E1   -57.691, E3 +134118.906}
ENDSPLINE

SPLINE
SPL {X  -111.648, Y  +797.871, Z    +0.000, E1   -60.847, E3 +134315.889}
SPL {X  -149.288, Y  +747.285, Z    +0.000, E1   -46.770, E3 +134311.879}
SPL {X  -161.496, Y  +712.364, Z    +0.000, E1   -31.137, E3 +134317.674}
SPL {X  -164.701, Y  +693.202, Z    +0.000, E1   -17.512, E3 +134316.649}
SPL {X  -165.453, Y  +683.578, Z    +0.000, E1    -9.445, E3 +134315.850}
SPL {X  -165.642, Y  +677.105, Z    +0.000, E1    -3.559, E3 +134316.161}
SPL {X  -165.650, Y  +673.263, Z    +0.000, E1    +0.216, E3 +134314.921}
SPL {X  -165.650, Y  +670.095, Z    +0.000, E1    +6.482, E3 +134314.325}
SPL {X  -165.650, Y  +666.485, Z    +0.000, E1   +14.169, E3 +134314.223}
SPL {X  -165.650, Y  +661.236, Z    +0.000, E1   +26.072, E3 +134313.913}
SPL {X  -165.650, Y  +653.063, Z    +0.000, E1   +42.395, E3 +134313.317}
SPL {X  -165.650, Y  +640.535, Z    +0.000, E1   +60.776, E3 +134310.801}
SPL {X  -165.650, Y  +618.963, Z    +0.000, E1   +72.815, E3 +134310.780}
SPL {X  -165.650, Y  +575.208, Z    +0.000, E1   +76.222, E3 +134322.041}
SPL {X  -165.650, Y  +394.754, Z    +0.000, E1   +73.248, E3 +134417.188}
ENDSPLINE

SPLINE
SPL {X  -165.650, Y  +407.500, Z    +0.000, E1   +70.919, E3 +134431.809}
ENDSPLINE

SPLINE
SPL {X  -165.650, Y  +390.855, Z    +0.000, E1   +71.004, E3 +134442.737}
SPL {X  -165.534, Y  +372.295, Z    +0.000, E1   +71.066, E3 +134455.287}
SPL {X  -164.687, Y  +360.663, Z    +0.000, E1   +70.826, E3 +134465.579}
SPL {X  -162.841, Y  +348.123, Z    +0.000, E1   +70.683, E3 +134475.958}
SPL {X  -162.352, Y  +345.609, Z    +0.000, E1   +69.290, E3 +134489.911}
SPL {X  -157.663, Y  +327.685, Z    +0.000, E1   +69.808, E3 +134498.771}
SPL {X  -152.892, Y  +314.750, Z    +0.000, E1   +69.675, E3 +134508.986}
SPL {X  -149.246, Y  +306.628, Z    +0.000, E1   +69.029, E3 +134519.455}
SPL {X  -145.495, Y  +299.310, Z    +0.000, E1   +68.659, E3 +134527.063}
SPL {X  -141.249, Y  +291.963, Z    +0.000, E1   +68.223, E3 +134535.044}
SPL {X  -137.649, Y  +286.345, Z    +0.000, E1   +67.498, E3 +134542.980}
SPL {X  -134.450, Y  +281.737, Z    +0.000, E1   +67.268, E3 +134547.370}
SPL {X  -131.812, Y  +278.173, Z    +0.000, E1   +66.669, E3 +134552.718}
SPL {X  -128.148, Y  +273.533, Z    +0.000, E1   +67.328, E3 +134553.077}
SPL {X  -116.216, Y  +260.459, Z    +0.000, E1   +70.200, E3 +134549.383}
SPL {X   -66.125, Y  +226.621, Z    +0.000, E1   +55.862, E3 +134712.282}
ENDSPLINE

SPLINE
SPL {X  -111.531, Y  +256.023, Z    +0.000, E1   +58.853, E3 +134855.163}
SPL {X  -139.240, Y  +288.767, Z    +0.000, E1   +52.898, E3 +134865.336}
SPL {X  -156.827, Y  +325.161, Z    +0.000, E1   +39.042, E3 +134863.706}
SPL {X  -162.324, Y  +345.471, Z    +0.000, E1   +27.849, E3 +134864.174}
SPL {X  -165.055, Y  +364.477, Z    +0.000, E1   +14.326, E3 +134864.612}
SPL {X  -165.646, Y  +377.353, Z    +0.000, E1    +3.112, E3 +134863.569}
SPL {X  -165.650, Y  +380.500, Z    +0.000, E1    -0.000, E3 +134862.695}
SPL {X  -165.650, Y  +381.828, Z    +0.000, E1    -2.219, E3 +134862.148}
SPL {X  -165.650, Y  +385.044, Z    +0.000, E1    -8.496, E3 +134861.947}
SPL {X  -165.650, Y  +388.717, Z    +0.000, E1   -16.400, E3 +134861.803}
SPL {X  -165.650, Y  +394.613, Z    +0.000, E1   -29.184, E3 +134861.272}
SPL {X  -165.650, Y  +402.836, Z    +0.000, E1   -44.797, E3 +134860.674}
SPL {X  -165.650, Y  +416.111, Z    +0.000, E1   -60.729, E3 +134859.741}
SPL {X  -165.650, Y  +471.994, Z    +0.000, E1   -75.670, E3 +134867.794}
SPL {X  -164.204, Y  +697.342, Z    +0.000, E1   -76.015, E3 +134955.817}
ENDSPLINE

SPLINE
SPL {X  -165.650, Y  +656.030, Z    +0.000, E1   -71.686, E3 +134977.257}
ENDSPLINE

SPLINE
SPL {X  -165.610, Y  +679.119, Z    +0.000, E1   -71.889, E3 +134990.880}
SPL {X  -164.561, Y  +694.465, Z    +0.000, E1   -71.736, E3 +135002.513}
SPL {X  -162.089, Y  +709.665, Z    +0.000, E1   -71.739, E3 +135012.714}
SPL {X  -159.776, Y  +719.221, Z    +0.000, E1   -71.038, E3 +135025.536}
SPL {X  -155.811, Y  +731.738, Z    +0.000, E1   -70.890, E3 +135035.224}
SPL {X  -152.643, Y  +739.844, Z    +0.000, E1   -70.463, E3 +135044.083}
SPL {X  -149.782, Y  +746.247, Z    +0.000, E1   -70.149, E3 +135050.773}
SPL {X  -146.450, Y  +752.910, Z    +0.000, E1   -69.680, E3 +135058.651}
SPL {X  -143.017, Y  +759.082, Z    +0.000, E1   -69.156, E3 +135066.262}
SPL {X  -140.057, Y  +763.953, Z    +0.000, E1   -68.829, E3 +135071.502}
SPL {X  -136.535, Y  +769.298, Z    +0.000, E1   -68.442, E3 +135077.363}
SPL {X  -133.553, Y  +773.498, Z    +0.000, E1   -67.773, E3 +135083.528}
SPL {X  -129.830, Y  +778.379, Z    +0.000, E1   -67.491, E3 +135088.154}
SPL {X  -116.788, Y  +792.975, Z    +0.000, E1   -71.297, E3 +135081.538}
SPL {X   -64.927, Y  +827.895, Z    +0.000, E1   -57.691, E3 +135207.141}
ENDSPLINE

SPLINE
SPL {X  -111.648, Y  +797.871, Z    +0.000, E1   -60.847, E3 +135404.124}
SPL {X  -149.288, Y  +747.285, Z    +0.000, E1   -46.770, E3 +135400.115}
SPL {X  -159.627, Y  +719.761, Z    +0.000, E1   -35.247, E3 +135405.180}
SPL {X  -164.185, Y  +697.485, Z    +0.000, E1   -20.950, E3 +135405.499}
SPL {X  -165.594, Y  +679.817, Z    +0.000, E1    -6.204, E3 +135404.275}
SPL {X  -165.650, Y  +673.522, Z    +0.000, E1    -0.038, E3 +135403.244}
SPL {X  -165.650, Y  +671.354, Z    +0.000, E1    +3.728, E3 +135402.732}
SPL {X  -165.650, Y  +666.485, Z    +0.000, E1   +14.169, E3 +135402.459}
SPL {X  -165.650, Y  +661.236, Z    +0.000, E1   +26.072, E3 +135402.148}
SPL {X  -165.650, Y  +653.063, Z    +0.000, E1   +42.395, E3 +135401.552}
SPL {X  -165.650, Y  +640.535, Z    +0.000, E1   +60.776, E3 +135399.037}
SPL {X  -165.650, Y  +618.963, Z    +0.000, E1   +72.815, E3 +135399.016}
SPL {X  -165.650, Y  +582.897, Z    +0.000, E1   +76.147, E3 +135407.677}
SPL {X  -165.650, Y  +558.388, Z    +0.000, E1   +76.294, E3 +135415.989}
SPL {X  -165.650, Y  +391.690, Z    +0.000, E1   +75.504, E3 +135485.755}
ENDSPLINE

SPLINE
SPL {X  -165.650, Y  +396.283, Z    +0.000, E1   +72.775, E3 +135509.060}
SPL {X  -165.650, Y  +407.500, Z    +0.000, E1   +70.919, E3 +135520.044}
ENDSPLINE

SPLINE
SPL {X  -165.650, Y  +390.855, Z    +0.000, E1   +71.004, E3 +135530.972}
SPL {X  -165.534, Y  +372.295, Z    +0.000, E1   +71.066, E3 +135543.522}
SPL {X  -164.039, Y  +355.451, Z    +0.000, E1   +70.703, E3 +135558.920}
SPL {X  -161.297, Y  +340.777, Z    +0.000, E1   +70.794, E3 +135568.213}
ENDSPLINE

SPLINE
SPL {X  -162.352, Y  +345.609, Z    +0.000, E1   +69.290, E3 +135578.146}
ENDSPLINE

SPLINE
SPL {X  -159.253, Y  +332.909, Z    +0.000, E1   +69.652, E3 +135584.492}
SPL {X  -155.267, Y  +320.775, Z    +0.000, E1   +69.854, E3 +135591.586}
SPL {X  -151.256, Y  +310.961, Z    +0.000, E1   +69.467, E3 +135601.461}
SPL {X  -148.628, Y  +305.359, Z    +0.000, E1   +68.848, E3 +135609.739}
SPL {X  -145.495, Y  +299.310, Z    +0.000, E1   +68.659, E3 +135615.299}
SPL {X  -142.111, Y  +293.387, Z    +0.000, E1   +68.421, E3 +135620.940}
SPL {X  -138.525, Y  +287.667, Z    +0.000, E1   +67.662, E3 +135629.500}
SPL {X  -134.450, Y  +281.737, Z    +0.000, E1   +67.268, E3 +135635.605}
SPL {X  -131.812, Y  +278.173, Z    +0.000, E1   +66.669, E3 +135640.954}
SPL {X  -128.148, Y  +273.533, Z    +0.000, E1   +67.328, E3 +135641.312}
SPL {X  -116.216, Y  +260.459, Z    +0.000, E1   +70.200, E3 +135637.619}
SPL {X   -66.125, Y  +226.621, Z    +0.000, E1   +55.862, E3 +135800.517}
ENDSPLINE

SPLINE
SPL {X  -111.531, Y  +256.023, Z    +0.000, E1   +58.853, E3 +135943.399}
SPL {X  -139.240, Y  +288.767, Z    +0.000, E1   +52.898, E3 +135953.572}
SPL {X  -156.827, Y  +325.161, Z    +0.000, E1   +39.042, E3 +135951.941}
SPL {X  -162.324, Y  +345.471, Z    +0.000, E1   +27.849, E3 +135952.410}
SPL {X  -165.055, Y  +364.477, Z    +0.000, E1   +14.326, E3 +135952.848}
SPL {X  -165.646, Y  +377.353, Z    +0.000, E1    +3.112, E3 +135951.805}
SPL {X  -165.650, Y  +380.500, Z    +0.000, E1    -0.000, E3 +135950.931}
SPL {X  -165.650, Y  +381.828, Z    +0.000, E1    -2.219, E3 +135950.383}
SPL {X  -165.650, Y  +385.044, Z    +0.000, E1    -8.496, E3 +135950.183}
SPL {X  -165.650, Y  +388.717, Z    +0.000, E1   -16.400, E3 +135950.038}
SPL {X  -165.650, Y  +394.613, Z    +0.000, E1   -29.184, E3 +135949.507}
SPL {X  -165.650, Y  +402.836, Z    +0.000, E1   -44.797, E3 +135948.910}
SPL {X  -165.650, Y  +416.111, Z    +0.000, E1   -60.729, E3 +135947.976}
SPL {X  -165.650, Y  +471.994, Z    +0.000, E1   -75.670, E3 +135956.030}
SPL {X  -164.204, Y  +697.342, Z    +0.000, E1   -76.015, E3 +136044.052}
ENDSPLINE

SPLINE
SPL {X  -165.650, Y  +656.030, Z    +0.000, E1   -71.686, E3 +136065.492}
ENDSPLINE

SPLINE
SPL {X  -165.610, Y  +679.119, Z    +0.000, E1   -71.889, E3 +136079.115}
SPL {X  -164.561, Y  +694.465, Z    +0.000, E1   -71.736, E3 +136090.748}
SPL {X  -162.089, Y  +709.665, Z    +0.000, E1   -71.739, E3 +136100.949}
SPL {X  -159.776, Y  +719.221, Z    +0.000, E1   -71.038, E3 +136113.771}
SPL {X  -155.811, Y  +731.738, Z    +0.000, E1   -70.890, E3 +136123.459}
SPL {X  -152.643, Y  +739.844, Z    +0.000, E1   -70.463, E3 +136132.319}
SPL {X  -149.782, Y  +746.247, Z    +0.000, E1   -70.149, E3 +136139.008}
SPL {X  -146.450, Y  +752.910, Z    +0.000, E1   -69.680, E3 +136146.886}
SPL {X  -143.017, Y  +759.082, Z    +0.000, E1   -69.156, E3 +136154.498}
SPL {X  -139.030, Y  +765.558, Z    +0.000, E1   -68.719, E3 +136161.531}
SPL {X  -135.682, Y  +770.527, Z    +0.000, E1   -68.337, E3 +136166.914}
SPL {X  -132.359, Y  +775.105, Z    +0.000, E1   -67.661, E3 +136173.456}
SPL {X  -128.720, Y  +779.765, Z    +0.000, E1   -67.454, E3 +136177.437}
SPL {X  -116.788, Y  +792.975, Z    +0.000, E1   -71.297, E3 +136169.774}
SPL {X   -64.927, Y  +827.895, Z    +0.000, E1   -57.691, E3 +136295.377}
ENDSPLINE

SPLINE
SPL {X  -111.648, Y  +797.871, Z    +0.000, E1   -60.847, E3 +136492.359}
SPL {X  -149.288, Y  +747.285, Z    +0.000, E1   -46.770, E3 +136488.350}
SPL {X  -159.627, Y  +719.761, Z    +0.000, E1   -35.247, E3 +136493.415}
SPL {X  -164.185, Y  +697.485, Z    +0.000, E1   -20.950, E3 +136493.734}
SPL {X  -165.594, Y  +679.817, Z    +0.000, E1    -6.204, E3 +136492.510}
SPL {X  -165.650, Y  +673.522, Z    +0.000, E1    -0.038, E3 +136491.479}
SPL {X  -165.650, Y  +671.354, Z    +0.000, E1    +3.728, E3 +136490.967}
SPL {X  -165.650, Y  +666.485, Z    +0.000, E1   +14.169, E3 +136490.694}
SPL {X  -165.650, Y  +661.236, Z    +0.000, E1   +26.072, E3 +136490.383}
SPL {X  -165.650, Y  +653.063, Z    +0.000, E1   +42.395, E3 +136489.787}
SPL {X  -165.650, Y  +640.535, Z    +0.000, E1   +60.776, E3 +136487.272}
SPL {X  -165.650, Y  +618.963, Z    +0.000, E1   +72.815, E3 +136487.251}
SPL {X  -165.650, Y  +575.208, Z    +0.000, E1   +76.222, E3 +136498.512}
SPL {X  -165.650, Y  +394.754, Z    +0.000, E1   +73.248, E3 +136593.658}
ENDSPLINE

SPLINE
SPL {X  -165.650, Y  +407.500, Z    +0.000, E1   +70.919, E3 +136608.279}
ENDSPLINE

SPLINE
SPL {X  -165.650, Y  +390.855, Z    +0.000, E1   +71.004, E3 +136619.207}
SPL {X  -165.534, Y  +372.295, Z    +0.000, E1   +71.066, E3 +136631.758}
SPL {X  -164.039, Y  +355.451, Z    +0.000, E1   +70.703, E3 +136647.156}
SPL {X  -161.297, Y  +340.777, Z    +0.000, E1   +70.794, E3 +136656.448}
ENDSPLINE

SPLINE
SPL {X  -162.352, Y  +345.609, Z    +0.000, E1   +69.290, E3 +136666.381}
ENDSPLINE

SPLINE
SPL {X  -159.253, Y  +332.909, Z    +0.000, E1   +69.652, E3 +136672.728}
SPL {X  -155.267, Y  +320.775, Z    +0.000, E1   +69.854, E3 +136679.821}
SPL {X  -151.256, Y  +310.961, Z    +0.000, E1   +69.467, E3 +136689.696}
SPL {X  -148.628, Y  +305.359, Z    +0.000, E1   +68.848, E3 +136697.974}
SPL {X  -145.495, Y  +299.310, Z    +0.000, E1   +68.659, E3 +136703.534}
SPL {X  -142.111, Y  +293.387, Z    +0.000, E1   +68.421, E3 +136709.175}
SPL {X  -138.525, Y  +287.667, Z    +0.000, E1   +67.662, E3 +136717.735}
SPL {X  -134.450, Y  +281.737, Z    +0.000, E1   +67.268, E3 +136723.840}
SPL {X  -131.812, Y  +278.173, Z    +0.000, E1   +66.669, E3 +136729.189}
SPL {X  -128.148, Y  +273.533, Z    +0.000, E1   +67.328, E3 +136729.547}
SPL {X  -116.216, Y  +260.459, Z    +0.000, E1   +70.200, E3 +136725.854}
SPL {X   -66.125, Y  +226.621, Z    +0.000, E1   +55.862, E3 +136888.752}
ENDSPLINE

SPLINE
SPL {X  -111.531, Y  +256.023, Z    +0.000, E1   +58.853, E3 +137031.634}
SPL {X  -139.240, Y  +288.767, Z    +0.000, E1   +52.898, E3 +137041.807}
SPL {X  -156.827, Y  +325.161, Z    +0.000, E1   +39.042, E3 +137040.176}
SPL {X  -162.324, Y  +345.471, Z    +0.000, E1   +27.849, E3 +137040.645}
SPL {X  -164.696, Y  +360.744, Z    +0.000, E1   +17.229, E3 +137041.559}
SPL {X  -165.561, Y  +373.081, Z    +0.000, E1    +6.973, E3 +137040.303}
SPL {X  -165.650, Y  +380.392, Z    +0.000, E1    +0.180, E3 +137039.220}
SPL {X  -165.650, Y  +381.828, Z    +0.000, E1    -2.219, E3 +137038.618}
SPL {X  -165.650, Y  +385.044, Z    +0.000, E1    -8.496, E3 +137038.418}
SPL {X  -165.650, Y  +390.492, Z    +0.000, E1   -20.084, E3 +137038.072}
SPL {X  -165.650, Y  +400.081, Z    +0.000, E1   -39.836, E3 +137037.377}
SPL {X  -165.650, Y  +416.111, Z    +0.000, E1   -60.729, E3 +137036.212}
SPL {X  -165.650, Y  +471.994, Z    +0.000, E1   -75.670, E3 +137044.265}
SPL {X  -164.204, Y  +697.342, Z    +0.000, E1   -76.015, E3 +137132.288}
ENDSPLINE

SPLINE
SPL {X  -165.650, Y  +664.340, Z    +0.000, E1   -71.862, E3 +137157.691}
ENDSPLINE

SPLINE
SPL {X  -165.116, Y  +688.792, Z    +0.000, E1   -71.759, E3 +137175.131}
SPL {X  -162.089, Y  +709.665, Z    +0.000, E1   -71.739, E3 +137189.184}
SPL {X  -160.450, Y  +716.681, Z    +0.000, E1   -71.166, E3 +137198.987}
SPL {X  -159.124, Y  +721.538, Z    +0.000, E1   -70.872, E3 +137204.914}
SPL {X  -155.811, Y  +731.738, Z    +0.000, E1   -70.890, E3 +137211.695}
SPL {X  -152.643, Y  +739.844, Z    +0.000, E1   -70.463, E3 +137220.554}
SPL {X  -149.782, Y  +746.247, Z    +0.000, E1   -70.149, E3 +137227.244}
SPL {X  -146.450, Y  +752.910, Z    +0.000, E1   -69.680, E3 +137235.122}
SPL {X  -143.017, Y  +759.082, Z    +0.000, E1   -69.156, E3 +137242.733}
SPL {X  -140.057, Y  +763.953, Z    +0.000, E1   -68.829, E3 +137247.972}
SPL {X  -136.535, Y  +769.298, Z    +0.000, E1   -68.442, E3 +137253.834}
SPL {X  -133.553, Y  +773.498, Z    +0.000, E1   -67.773, E3 +137259.999}
SPL {X  -129.830, Y  +778.379, Z    +0.000, E1   -67.491, E3 +137264.625}
SPL {X  -116.788, Y  +792.975, Z    +0.000, E1   -71.297, E3 +137258.009}
SPL {X   -64.927, Y  +827.895, Z    +0.000, E1   -57.691, E3 +137383.612}
ENDSPLINE

SPLINE
SPL {X  -111.648, Y  +797.871, Z    +0.000, E1   -60.847, E3 +137580.594}
SPL {X  -149.288, Y  +747.285, Z    +0.000, E1   -46.770, E3 +137576.585}
SPL {X  -159.627, Y  +719.761, Z    +0.000, E1   -35.247, E3 +137581.650}
SPL {X  -164.185, Y  +697.485, Z    +0.000, E1   -20.950, E3 +137581.969}
SPL {X  -165.594, Y  +679.817, Z    +0.000, E1    -6.204, E3 +137580.746}
SPL {X  -165.650, Y  +673.522, Z    +0.000, E1    -0.038, E3 +137579.715}
SPL {X  -165.650, Y  +671.354, Z    +0.000, E1    +3.728, E3 +137579.202}
SPL {X  -165.650, Y  +666.485, Z    +0.000, E1   +14.169, E3 +137578.929}
SPL {X  -165.650, Y  +661.236, Z    +0.000, E1   +26.072, E3 +137578.618}
SPL {X  -165.650, Y  +653.063, Z    +0.000, E1   +42.395, E3 +137578.023}
SPL {X  -165.650, Y  +640.535, Z    +0.000, E1   +60.776, E3 +137575.507}
SPL {X  -165.650, Y  +618.963, Z    +0.000, E1   +72.815, E3 +137575.486}
SPL {X  -165.650, Y  +575.208, Z    +0.000, E1   +76.222, E3 +137586.747}
SPL {X  -165.650, Y  +394.754, Z    +0.000, E1   +73.248, E3 +137681.894}
ENDSPLINE

SPLINE
SPL {X  -165.650, Y  +407.500, Z    +0.000, E1   +70.919, E3 +137696.515}
ENDSPLINE

SPLINE
SPL {X  -165.650, Y  +390.855, Z    +0.000, E1   +71.004, E3 +137707.442}
SPL {X  -165.534, Y  +372.295, Z    +0.000, E1   +71.066, E3 +137719.993}
SPL {X  -164.039, Y  +355.451, Z    +0.000, E1   +70.703, E3 +137735.391}
SPL {X  -161.297, Y  +340.777, Z    +0.000, E1   +70.794, E3 +137744.683}
ENDSPLINE

SPLINE
SPL {X  -162.352, Y  +345.609, Z    +0.000, E1   +69.290, E3 +137754.617}
ENDSPLINE

SPLINE
SPL {X  -157.663, Y  +327.685, Z    +0.000, E1   +69.808, E3 +137763.477}
SPL {X  -152.892, Y  +314.750, Z    +0.000, E1   +69.675, E3 +137773.692}
SPL {X  -149.246, Y  +306.628, Z    +0.000, E1   +69.029, E3 +137784.161}
SPL {X  -145.495, Y  +299.310, Z    +0.000, E1   +68.659, E3 +137791.769}
SPL {X  -142.111, Y  +293.387, Z    +0.000, E1   +68.421, E3 +137797.411}
SPL {X  -138.525, Y  +287.667, Z    +0.000, E1   +67.662, E3 +137805.970}
SPL {X  -134.450, Y  +281.737, Z    +0.000, E1   +67.268, E3 +137812.076}
SPL {X  -131.812, Y  +278.173, Z    +0.000, E1   +66.669, E3 +137817.424}
SPL {X  -128.148, Y  +273.533, Z    +0.000, E1   +67.328, E3 +137817.783}
SPL {X  -116.216, Y  +260.459, Z    +0.000, E1   +70.200, E3 +137814.089}
SPL {X   -66.125, Y  +226.621, Z    +0.000, E1   +55.862, E3 +137976.987}
ENDSPLINE

SPLINE
SPL {X  -111.531, Y  +256.023, Z    +0.000, E1   +58.853, E3 +138119.869}
SPL {X  -139.240, Y  +288.767, Z    +0.000, E1   +52.898, E3 +138130.042}
SPL {X  -156.827, Y  +325.161, Z    +0.000, E1   +39.042, E3 +138128.412}
SPL {X  -162.324, Y  +345.471, Z    +0.000, E1   +27.849, E3 +138128.880}
SPL {X  -165.055, Y  +364.477, Z    +0.000, E1   +14.326, E3 +138129.318}
SPL {X  -165.646, Y  +377.353, Z    +0.000, E1    +3.112, E3 +138128.275}
SPL {X  -165.650, Y  +380.500, Z    +0.000, E1    -0.000, E3 +138127.401}
SPL {X  -165.650, Y  +381.828, Z    +0.000, E1    -2.219, E3 +138126.853}
SPL {X  -165.650, Y  +385.044, Z    +0.000, E1    -8.496, E3 +138126.653}
SPL {X  -165.650, Y  +390.492, Z    +0.000, E1   -20.084, E3 +138126.307}
SPL {X  -165.650, Y  +400.081, Z    +0.000, E1   -39.836, E3 +138125.613}
SPL {X  -165.650, Y  +416.111, Z    +0.000, E1   -60.729, E3 +138124.447}
SPL {X  -165.650, Y  +471.994, Z    +0.000, E1   -75.670, E3 +138132.500}
SPL {X  -164.204, Y  +697.342, Z    +0.000, E1   -76.015, E3 +138220.523}
ENDSPLINE

SPLINE
SPL {X  -165.650, Y  +664.340, Z    +0.000, E1   -71.862, E3 +138245.927}
ENDSPLINE

SPLINE
SPL {X  -165.116, Y  +688.792, Z    +0.000, E1   -71.759, E3 +138263.366}
SPL {X  -162.089, Y  +709.665, Z    +0.000, E1   -71.739, E3 +138277.420}
SPL {X  -160.450, Y  +716.681, Z    +0.000, E1   -71.166, E3 +138287.223}
SPL {X  -159.124, Y  +721.538, Z    +0.000, E1   -70.872, E3 +138293.150}
SPL {X  -155.811, Y  +731.738, Z    +0.000, E1   -70.890, E3 +138299.930}
SPL {X  -152.643, Y  +739.844, Z    +0.000, E1   -70.463, E3 +138308.789}
SPL {X  -149.782, Y  +746.247, Z    +0.000, E1   -70.149, E3 +138315.479}
SPL {X  -146.450, Y  +752.910, Z    +0.000, E1   -69.680, E3 +138323.357}
SPL {X  -143.017, Y  +759.082, Z    +0.000, E1   -69.156, E3 +138330.968}
SPL {X  -139.030, Y  +765.558, Z    +0.000, E1   -68.719, E3 +138338.001}
SPL {X  -135.682, Y  +770.527, Z    +0.000, E1   -68.337, E3 +138343.385}
SPL {X  -132.359, Y  +775.105, Z    +0.000, E1   -67.661, E3 +138349.927}
SPL {X  -128.720, Y  +779.765, Z    +0.000, E1   -67.454, E3 +138353.908}
SPL {X  -116.788, Y  +792.975, Z    +0.000, E1   -71.297, E3 +138346.244}
SPL {X   -64.927, Y  +827.895, Z    +0.000, E1   -57.691, E3 +138471.847}
ENDSPLINE

SPLINE
SPL {X  -111.648, Y  +797.871, Z    +0.000, E1   -60.847, E3 +138668.830}
SPL {X  -149.288, Y  +747.285, Z    +0.000, E1   -46.770, E3 +138664.820}
SPL {X  -161.496, Y  +712.364, Z    +0.000, E1   -31.137, E3 +138670.616}
SPL {X  -164.701, Y  +693.202, Z    +0.000, E1   -17.512, E3 +138669.590}
SPL {X  -165.594, Y  +679.817, Z    +0.000, E1    -6.204, E3 +138668.981}
SPL {X  -165.650, Y  +673.522, Z    +0.000, E1    -0.038, E3 +138667.950}
SPL {X  -165.650, Y  +671.354, Z    +0.000, E1    +3.728, E3 +138667.437}
SPL {X  -165.650, Y  +666.485, Z    +0.000, E1   +14.169, E3 +138667.165}
SPL {X  -165.650, Y  +661.236, Z    +0.000, E1   +26.072, E3 +138666.854}
SPL {X  -165.650, Y  +653.063, Z    +0.000, E1   +42.395, E3 +138666.258}
SPL {X  -165.650, Y  +640.535, Z    +0.000, E1   +60.776, E3 +138663.743}
SPL {X  -165.650, Y  +618.963, Z    +0.000, E1   +72.815, E3 +138663.722}
SPL {X  -165.650, Y  +575.208, Z    +0.000, E1   +76.222, E3 +138674.982}
SPL {X  -165.650, Y  +394.754, Z    +0.000, E1   +73.248, E3 +138770.129}
ENDSPLINE

SPLINE
SPL {X  -165.650, Y  +407.500, Z    +0.000, E1   +70.919, E3 +138784.750}
ENDSPLINE

SPLINE
SPL {X  -165.650, Y  +390.855, Z    +0.000, E1   +71.004, E3 +138795.678}
SPL {X  -165.534, Y  +372.295, Z    +0.000, E1   +71.066, E3 +138808.228}
SPL {X  -164.039, Y  +355.451, Z    +0.000, E1   +70.703, E3 +138823.626}
SPL {X  -161.297, Y  +340.777, Z    +0.000, E1   +70.794, E3 +138832.919}
ENDSPLINE

SPLINE
SPL {X  -162.352, Y  +345.609, Z    +0.000, E1   +69.290, E3 +138842.852}
ENDSPLINE

SPLINE
SPL {X  -157.663, Y  +327.685, Z    +0.000, E1   +69.808, E3 +138851.712}
SPL {X  -152.892, Y  +314.750, Z    +0.000, E1   +69.675, E3 +138861.928}
SPL {X  -149.246, Y  +306.628, Z    +0.000, E1   +69.029, E3 +138872.396}
SPL {X  -145.495, Y  +299.310, Z    +0.000, E1   +68.659, E3 +138880.004}
SPL {X  -142.111, Y  +293.387, Z    +0.000, E1   +68.421, E3 +138885.646}
SPL {X  -138.525, Y  +287.667, Z    +0.000, E1   +67.662, E3 +138894.206}
SPL {X  -134.450, Y  +281.737, Z    +0.000, E1   +67.268, E3 +138900.311}
SPL {X  -131.812, Y  +278.173, Z    +0.000, E1   +66.669, E3 +138905.660}
SPL {X  -128.148, Y  +273.533, Z    +0.000, E1   +67.328, E3 +138906.018}
SPL {X  -116.216, Y  +260.459, Z    +0.000, E1   +70.200, E3 +138902.325}
SPL {X   -66.125, Y  +226.621, Z    +0.000, E1   +55.862, E3 +139065.223}
ENDSPLINE

SPLINE
SPL {X  -111.531, Y  +256.023, Z    +0.000, E1   +58.853, E3 +139208.105}
SPL {X  -139.240, Y  +288.767, Z    +0.000, E1   +52.898, E3 +139218.277}
SPL {X  -156.827, Y  +325.161, Z    +0.000, E1   +39.042, E3 +139216.647}
SPL {X  -162.324, Y  +345.471, Z    +0.000, E1   +27.849, E3 +139217.115}
SPL {X  -164.696, Y  +360.744, Z    +0.000, E1   +17.229, E3 +139218.030}
SPL {X  -165.561, Y  +373.081, Z    +0.000, E1    +6.973, E3 +139216.774}
SPL {X  -165.650, Y  +380.800, Z    +0.000, E1    -0.199, E3 +139215.520}
SPL {X  -165.650, Y  +385.044, Z    +0.000, E1    -8.496, E3 +139214.888}
SPL {X  -165.650, Y  +390.492, Z    +0.000, E1   -20.084, E3 +139214.543}
SPL {X  -165.650, Y  +400.081, Z    +0.000, E1   -39.836, E3 +139213.848}
SPL {X  -165.650, Y  +416.111, Z    +0.000, E1   -60.729, E3 +139212.682}
SPL {X  -165.650, Y  +457.077, Z    +0.000, E1   -75.210, E3 +139216.006}
SPL {X  -165.650, Y  +475.293, Z    +0.000, E1   -75.741, E3 +139221.784}
SPL {X  -164.204, Y  +697.342, Z    +0.000, E1   -76.015, E3 +139308.758}
ENDSPLINE

SPLINE
SPL {X  -165.650, Y  +656.030, Z    +0.000, E1   -71.686, E3 +139330.198}
ENDSPLINE

SPLINE
SPL {X  -165.472, Y  +683.167, Z    +0.000, E1   -72.022, E3 +139345.206}
SPL {X  -163.865, Y  +699.752, Z    +0.000, E1   -71.643, E3 +139359.829}
SPL {X  -161.571, Y  +712.032, Z    +0.000, E1   -71.595, E3 +139368.422}
SPL {X  -159.776, Y  +719.221, Z    +0.000, E1   -71.038, E3 +139378.477}
SPL {X  -155.811, Y  +731.738, Z    +0.000, E1   -70.890, E3 +139388.165}
SPL {X  -152.643, Y  +739.844, Z    +0.000, E1   -70.463, E3 +139397.024}
SPL {X  -149.782, Y  +746.247, Z    +0.000, E1   -70.149, E3 +139403.714}
SPL {X  -146.450, Y  +752.910, Z    +0.000, E1   -69.680, E3 +139411.592}
SPL {X  -143.017, Y  +759.082, Z    +0.000, E1   -69.156, E3 +139419.204}
SPL {X  -139.030, Y  +765.558, Z    +0.000, E1   -68.719, E3 +139426.237}
SPL {X  -135.682, Y  +770.527, Z    +0.000, E1   -68.337, E3 +139431.620}
SPL {X  -132.359, Y  +775.105, Z    +0.000, E1   -67.661, E3 +139438.162}
SPL {X  -128.720, Y  +779.765, Z    +0.000, E1   -67.454, E3 +139442.143}
SPL {X  -116.788, Y  +792.975, Z    +0.000, E1   -71.297, E3 +139434.480}
SPL {X   -64.927, Y  +827.895, Z    +0.000, E1   -57.691, E3 +139560.083}
ENDSPLINE

SPLINE
SPL {X  -111.648, Y  +797.871, Z    +0.000, E1   -60.847, E3 +139757.065}
SPL {X  -149.288, Y  +747.285, Z    +0.000, E1   -46.770, E3 +139753.056}
SPL {X  -159.627, Y  +719.761, Z    +0.000, E1   -35.247, E3 +139758.121}
SPL {X  -164.185, Y  +697.485, Z    +0.000, E1   -20.950, E3 +139758.440}
SPL {X  -165.453, Y  +683.578, Z    +0.000, E1    -9.445, E3 +139757.027}
SPL {X  -165.642, Y  +677.105, Z    +0.000, E1    -3.559, E3 +139757.338}
SPL {X  -165.650, Y  +673.522, Z    +0.000, E1    -0.038, E3 +139756.185}
SPL {X  -165.650, Y  +671.354, Z    +0.000, E1    +3.728, E3 +139755.673}
SPL {X  -165.650, Y  +666.485, Z    +0.000, E1   +14.169, E3 +139755.400}
SPL {X  -165.650, Y  +661.236, Z    +0.000, E1   +26.072, E3 +139755.089}
SPL {X  -165.650, Y  +655.357, Z    +0.000, E1   +38.693, E3 +139754.317}
SPL {X  -165.650, Y  +646.637, Z    +0.000, E1   +52.169, E3 +139754.098}
SPL {X  -165.650, Y  +637.909, Z    +0.000, E1   +64.161, E3 +139750.894}
SPL {X  -165.650, Y  +618.963, Z    +0.000, E1   +72.815, E3 +139751.957}
SPL {X  -165.650, Y  +582.897, Z    +0.000, E1   +76.147, E3 +139760.618}
SPL {X  -165.650, Y  +558.388, Z    +0.000, E1   +76.294, E3 +139768.930}
SPL {X  -165.650, Y  +391.690, Z    +0.000, E1   +75.504, E3 +139838.697}
ENDSPLINE

SPLINE
SPL {X  -165.650, Y  +396.283, Z    +0.000, E1   +72.775, E3 +139862.002}
SPL {X  -165.650, Y  +407.500, Z    +0.000, E1   +70.919, E3 +139872.985}
ENDSPLINE

SPLINE
SPL {X  -165.650, Y  +384.687, Z    +0.000, E1   +71.028, E3 +139888.231}
SPL {X  -164.996, Y  +363.797, Z    +0.000, E1   +70.987, E3 +139903.206}
SPL {X  -162.841, Y  +348.123, Z    +0.000, E1   +70.683, E3 +139917.134}
SPL {X  -162.352, Y  +345.609, Z    +0.000, E1   +69.290, E3 +139931.087}
SPL {X  -157.663, Y  +327.685, Z    +0.000, E1   +69.808, E3 +139939.947}
SPL {X  -152.892, Y  +314.750, Z    +0.000, E1   +69.675, E3 +139950.163}
SPL {X  -149.246, Y  +306.628, Z    +0.000, E1   +69.029, E3 +139960.631}
SPL {X  -144.614, Y  +297.712, Z    +0.000, E1   +68.717, E3 +139968.985}
SPL {X  -141.011, Y  +291.576, Z    +0.000, E1   +68.040, E3 +139977.463}
SPL {X  -137.649, Y  +286.345, Z    +0.000, E1   +67.498, E3 +139984.156}
SPL {X  -134.450, Y  +281.737, Z    +0.000, E1   +67.268, E3 +139988.546}
SPL {X  -131.812, Y  +278.173, Z    +0.000, E1   +66.669, E3 +139993.895}
SPL {X  -128.148, Y  +273.533, Z    +0.000, E1   +67.328, E3 +139994.253}
SPL {X  -116.216, Y  +260.459, Z    +0.000, E1   +70.200, E3 +139990.560}
SPL {X   -66.125, Y  +226.621, Z    +0.000, E1   +55.862, E3 +140153.458}
ENDSPLINE

SPLINE
SPL {X  -111.531, Y  +256.023, Z    +0.000, E1   +58.853, E3 +140296.340}
SPL {X  -139.240, Y  +288.767, Z    +0.000, E1   +52.898, E3 +140306.513}
SPL {X  -156.827, Y  +325.161, Z    +0.000, E1   +39.042, E3 +140304.882}
SPL {X  -162.324, Y  +345.471, Z    +0.000, E1   +27.849, E3 +140305.351}
SPL {X  -165.055, Y  +364.477, Z    +0.000, E1   +14.326, E3 +140305.789}
SPL {X  -165.646, Y  +377.353, Z    +0.000, E1    +3.112, E3 +140304.746}
SPL {X  -165.650, Y  +380.899, Z    +0.000, E1    -0.394, E3 +140303.707}
SPL {X  -165.650, Y  +385.044, Z    +0.000, E1    -8.496, E3 +140303.124}
SPL {X  -165.650, Y  +390.492, Z    +0.000, E1   -20.084, E3 +140302.778}
SPL {X  -165.650, Y  +398.793, Z    +0.000, E1   -37.509, E3 +140302.296}
SPL {X  -165.650, Y  +409.325, Z    +0.000, E1   -54.181, E3 +140300.976}
SPL {X  -165.650, Y  +420.423, Z    +0.000, E1   -63.808, E3 +140301.125}
SPL {X  -165.650, Y  +471.994, Z    +0.000, E1   -75.670, E3 +140308.971}
SPL {X  -164.204, Y  +697.342, Z    +0.000, E1   -76.015, E3 +140396.994}
ENDSPLINE

SPLINE
SPL {X  -165.650, Y  +664.340, Z    +0.000, E1   -71.862, E3 +140422.397}
ENDSPLINE

SPLINE
SPL {X  -165.237, Y  +687.187, Z    +0.000, E1   -71.947, E3 +140436.659}
SPL {X  -163.865, Y  +699.752, Z    +0.000, E1   -71.643, E3 +140448.064}
SPL {X  -161.041, Y  +714.304, Z    +0.000, E1   -71.423, E3 +140459.968}
SPL {X  -159.124, Y  +721.538, Z    +0.000, E1   -70.872, E3 +140469.620}
SPL {X  -155.811, Y  +731.738, Z    +0.000, E1   -70.890, E3 +140476.401}
SPL {X  -152.643, Y  +739.844, Z    +0.000, E1   -70.463, E3 +140485.260}
SPL {X  -149.782, Y  +746.247, Z    +0.000, E1   -70.149, E3 +140491.950}
SPL {X  -146.450, Y  +752.910, Z    +0.000, E1   -69.680, E3 +140499.828}
SPL {X  -143.017, Y  +759.082, Z    +0.000, E1   -69.156, E3 +140507.439}
SPL {X  -140.057, Y  +763.953, Z    +0.000, E1   -68.829, E3 +140512.678}
SPL {X  -136.535, Y  +769.298, Z    +0.000, E1   -68.442, E3 +140518.540}
SPL {X  -133.553, Y  +773.498, Z    +0.000, E1   -67.773, E3 +140524.705}
SPL {X  -129.830, Y  +778.379, Z    +0.000, E1   -67.491, E3 +140529.331}
SPL {X  -116.788, Y  +792.975, Z    +0.000, E1   -71.297, E3 +140522.715}
SPL {X   -64.927, Y  +827.895, Z    +0.000, E1   -57.691, E3 +140648.318}
ENDSPLINE

SPLINE
SPL {X  -111.648, Y  +797.871, Z    +0.000, E1   -60.847, E3 +140845.300}
SPL {X  -149.288, Y  +747.285, Z    +0.000, E1   -46.770, E3 +140841.291}
SPL {X  -159.627, Y  +719.761, Z    +0.000, E1   -35.247, E3 +140846.356}
SPL {X  -164.185, Y  +697.485, Z    +0.000, E1   -20.950, E3 +140846.675}
SPL {X  -165.453, Y  +683.578, Z    +0.000, E1    -9.445, E3 +140845.262}
SPL {X  -165.642, Y  +677.105, Z    +0.000, E1    -3.559, E3 +140845.573}
SPL {X  -165.650, Y  +673.522, Z    +0.000, E1    -0.038, E3 +140844.420}
SPL {X  -165.650, Y  +671.354, Z    +0.000, E1    +3.728, E3 +140843.908}
SPL {X  -165.650, Y  +666.485, Z    +0.000, E1   +14.169, E3 +140843.635}
SPL {X  -165.650, Y  +661.236, Z    +0.000, E1   +26.072, E3 +140843.324}
SPL {X  -165.650, Y  +653.063, Z    +0.000, E1   +42.395, E3 +140842.728}
SPL {X  -165.650, Y  +640.535, Z    +0.000, E1   +60.776, E3 +140840.213}
SPL {X  -165.650, Y  +618.963, Z    +0.000, E1   +72.815, E3 +140840.192}
SPL {X  -165.650, Y  +575.208, Z    +0.000, E1   +76.222, E3 +140851.453}
SPL {X  -165.650, Y  +394.754, Z    +0.000, E1   +73.248, E3 +140946.599}
ENDSPLINE

SPLINE
SPL {X  -165.650, Y  +407.500, Z    +0.000, E1   +70.919, E3 +140961.221}
ENDSPLINE

SPLINE
SPL {X  -165.650, Y  +390.855, Z    +0.000, E1   +71.004, E3 +140972.148}
SPL {X  -165.534, Y  +372.295, Z    +0.000, E1   +71.066, E3 +140984.699}
SPL {X  -164.687, Y  +360.663, Z    +0.000, E1   +70.826, E3 +140994.990}
SPL {X  -162.841, Y  +348.123, Z    +0.000, E1   +70.683, E3 +141005.369}
SPL {X  -162.352, Y  +345.609, Z    +0.000, E1   +69.290, E3 +141019.322}
SPL {X  -159.253, Y  +332.909, Z    +0.000, E1   +69.652, E3 +141025.669}
SPL {X  -156.309, Y  +323.661, Z    +0.000, E1   +69.908, E3 +141030.183}
SPL {X  -152.892, Y  +314.750, Z    +0.000, E1   +69.675, E3 +141038.398}
SPL {X  -149.246, Y  +306.628, Z    +0.000, E1   +69.029, E3 +141048.866}
SPL {X  -145.495, Y  +299.310, Z    +0.000, E1   +68.659, E3 +141056.475}
SPL {X  -142.111, Y  +293.387, Z    +0.000, E1   +68.421, E3 +141062.117}
SPL {X  -138.525, Y  +287.667, Z    +0.000, E1   +67.662, E3 +141070.676}
SPL {X  -134.450, Y  +281.737, Z    +0.000, E1   +67.268, E3 +141076.782}
SPL {X  -131.812, Y  +278.173, Z    +0.000, E1   +66.669, E3 +141082.130}
SPL {X  -128.148, Y  +273.533, Z    +0.000, E1   +67.328, E3 +141082.489}
SPL {X  -116.216, Y  +260.459, Z    +0.000, E1   +70.200, E3 +141078.795}
SPL {X   -66.125, Y  +226.621, Z    +0.000, E1   +55.862, E3 +141241.693}
ENDSPLINE

SPLINE
SPL {X  -111.531, Y  +256.023, Z    +0.000, E1   +58.853, E3 +141384.575}
SPL {X  -139.240, Y  +288.767, Z    +0.000, E1   +52.898, E3 +141394.748}
SPL {X  -156.827, Y  +325.161, Z    +0.000, E1   +39.042, E3 +141393.117}
SPL {X  -163.133, Y  +349.734, Z    +0.000, E1   +25.193, E3 +141394.242}
SPL {X  -165.214, Y  +366.494, Z    +0.000, E1   +12.605, E3 +141393.715}
SPL {X  -165.615, Y  +375.073, Z    +0.000, E1    +5.133, E3 +141393.203}
SPL {X  -165.650, Y  +380.392, Z    +0.000, E1    +0.180, E3 +141392.161}
SPL {X  -165.650, Y  +381.828, Z    +0.000, E1    -2.219, E3 +141391.559}
SPL {X  -165.650, Y  +385.044, Z    +0.000, E1    -8.496, E3 +141391.359}
SPL {X  -165.650, Y  +388.717, Z    +0.000, E1   -16.400, E3 +141391.215}
SPL {X  -165.650, Y  +394.613, Z    +0.000, E1   -29.184, E3 +141390.684}
SPL {X  -165.650, Y  +402.836, Z    +0.000, E1   -44.797, E3 +141390.086}
SPL {X  -165.650, Y  +416.111, Z    +0.000, E1   -60.729, E3 +141389.153}
SPL {X  -165.650, Y  +471.994, Z    +0.000, E1   -75.670, E3 +141397.206}
SPL {X  -164.204, Y  +697.342, Z    +0.000, E1   -76.015, E3 +141485.229}
ENDSPLINE

SPLINE
SPL {X  -165.650, Y  +656.030, Z    +0.000, E1   -71.686, E3 +141506.668}
ENDSPLINE

SPLINE
SPL {X  -165.610, Y  +679.119, Z    +0.000, E1   -71.889, E3 +141520.292}
SPL {X  -164.561, Y  +694.465, Z    +0.000, E1   -71.736, E3 +141531.925}
SPL {X  -162.089, Y  +709.665, Z    +0.000, E1   -71.739, E3 +141542.126}
SPL {X  -159.776, Y  +719.221, Z    +0.000, E1   -71.038, E3 +141554.948}
SPL {X  -155.811, Y  +731.738, Z    +0.000, E1   -70.890, E3 +141564.636}
SPL {X  -152.643, Y  +739.844, Z    +0.000, E1   -70.463, E3 +141573.495}
SPL {X  -149.782, Y  +746.247, Z    +0.000, E1   -70.149, E3 +141580.185}
SPL {X  -146.450, Y  +752.910, Z    +0.000, E1   -69.680, E3 +141588.063}
SPL {X  -143.017, Y  +759.082, Z    +0.000, E1   -69.156, E3 +141595.674}
SPL {X  -139.030, Y  +765.558, Z    +0.000, E1   -68.719, E3 +141602.707}
SPL {X  -134.589, Y  +772.070, Z    +0.000, E1   -68.090, E3 +141610.556}
SPL {X  -129.830, Y  +778.379, Z    +0.000, E1   -67.491, E3 +141617.566}
SPL {X  -116.788, Y  +792.975, Z    +0.000, E1   -71.297, E3 +141610.950}
SPL {X   -64.927, Y  +827.895, Z    +0.000, E1   -57.691, E3 +141736.553}
ENDSPLINE

SPLINE
SPL {X  -111.648, Y  +797.871, Z    +0.000, E1   -60.847, E3 +141933.536}
SPL {X  -149.288, Y  +747.285, Z    +0.000, E1   -46.770, E3 +141929.526}
SPL {X  -159.627, Y  +719.761, Z    +0.000, E1   -35.247, E3 +141934.591}
SPL {X  -164.185, Y  +697.485, Z    +0.000, E1   -20.950, E3 +141934.910}
SPL {X  -165.453, Y  +683.578, Z    +0.000, E1    -9.445, E3 +141933.497}
SPL {X  -165.642, Y  +677.105, Z    +0.000, E1    -3.559, E3 +141933.808}
SPL {X  -165.650, Y  +673.263, Z    +0.000, E1    +0.216, E3 +141932.568}
SPL {X  -165.650, Y  +670.095, Z    +0.000, E1    +6.482, E3 +141931.972}
SPL {X  -165.650, Y  +666.485, Z    +0.000, E1   +14.169, E3 +141931.870}
SPL {X  -165.650, Y  +661.236, Z    +0.000, E1   +26.072, E3 +141931.560}
SPL {X  -165.650, Y  +653.063, Z    +0.000, E1   +42.395, E3 +141930.964}
SPL {X  -165.650, Y  +640.535, Z    +0.000, E1   +60.776, E3 +141928.449}
SPL {X  -165.650, Y  +618.963, Z    +0.000, E1   +72.815, E3 +141928.428}
SPL {X  -165.650, Y  +575.208, Z    +0.000, E1   +76.222, E3 +141939.688}
SPL {X  -165.650, Y  +394.754, Z    +0.000, E1   +73.248, E3 +142034.835}
ENDSPLINE

SPLINE
SPL {X  -165.650, Y  +407.500, Z    +0.000, E1   +70.919, E3 +142049.456}
ENDSPLINE

SPLINE
SPL {X  -165.650, Y  +390.855, Z    +0.000, E1   +71.004, E3 +142060.384}
SPL {X  -165.534, Y  +372.295, Z    +0.000, E1   +71.066, E3 +142072.934}
SPL {X  -164.687, Y  +360.663, Z    +0.000, E1   +70.826, E3 +142083.226}
SPL {X  -162.841, Y  +348.123, Z    +0.000, E1   +70.683, E3 +142093.605}
SPL {X  -162.352, Y  +345.609, Z    +0.000, E1   +69.290, E3 +142107.558}
SPL {X  -159.253, Y  +332.909, Z    +0.000, E1   +69.652, E3 +142113.904}
SPL {X  -156.309, Y  +323.661, Z    +0.000, E1   +69.908, E3 +142118.419}
SPL {X  -152.892, Y  +314.750, Z    +0.000, E1   +69.675, E3 +142126.634}
SPL {X  -149.246, Y  +306.628, Z    +0.000, E1   +69.029, E3 +142137.102}
SPL {X  -145.495, Y  +299.310, Z    +0.000, E1   +68.659, E3 +142144.710}
SPL {X  -141.249, Y  +291.963, Z    +0.000, E1   +68.223, E3 +142152.691}
SPL {X  -137.649, Y  +286.345, Z    +0.000, E1   +67.498, E3 +142160.627}
SPL {X  -134.450, Y  +281.737, Z    +0.000, E1   +67.268, E3 +142165.017}
SPL {X  -131.812, Y  +278.173, Z    +0.000, E1   +66.669, E3 +142170.365}
SPL {X  -128.148, Y  +273.533, Z    +0.000, E1   +67.328, E3 +142170.724}
SPL {X  -116.216, Y  +260.459, Z    +0.000, E1   +70.200, E3 +142167.030}
SPL {X   -66.125, Y  +226.621, Z    +0.000, E1   +55.862, E3 +142329.929}
ENDSPLINE

SPLINE
SPL {X  -111.531, Y  +256.023, Z    +0.000, E1   +58.853, E3 +142472.810}
SPL {X  -139.240, Y  +288.767, Z    +0.000, E1   +52.898, E3 +142482.983}
SPL {X  -156.827, Y  +325.161, Z    +0.000, E1   +39.042, E3 +142481.353}
SPL {X  -163.133, Y  +349.734, Z    +0.000, E1   +25.193, E3 +142482.477}
SPL {X  -165.214, Y  +366.494, Z    +0.000, E1   +12.605, E3 +142481.950}
SPL {X  -165.615, Y  +375.073, Z    +0.000, E1    +5.133, E3 +142481.438}
SPL {X  -165.650, Y  +380.800, Z    +0.000, E1    -0.199, E3 +142480.226}
SPL {X  -165.650, Y  +385.044, Z    +0.000, E1    -8.496, E3 +142479.594}
SPL {X  -165.650, Y  +390.492, Z    +0.000, E1   -20.084, E3 +142479.249}
SPL {X  -165.650, Y  +400.081, Z    +0.000, E1   -39.836, E3 +142478.554}
SPL {X  -165.650, Y  +416.111, Z    +0.000, E1   -60.729, E3 +142477.388}
SPL {X  -165.650, Y  +457.077, Z    +0.000, E1   -75.210, E3 +142480.712}
SPL {X  -165.650, Y  +475.293, Z    +0.000, E1   -75.741, E3 +142486.489}
SPL {X  -164.204, Y  +697.342, Z    +0.000, E1   -76.015, E3 +142573.464}
ENDSPLINE

SPLINE
SPL {X  -165.650, Y  +664.340, Z    +0.000, E1   -71.862, E3 +142598.868}
ENDSPLINE

SPLINE
SPL {X  -165.237, Y  +687.187, Z    +0.000, E1   -71.947, E3 +142613.129}
SPL {X  -163.865, Y  +699.752, Z    +0.000, E1   -71.643, E3 +142624.535}
SPL {X  -161.821, Y  +710.908, Z    +0.000, E1   -71.322, E3 +142635.075}
SPL {X  -158.993, Y  +721.987, Z    +0.000, E1   -71.173, E3 +142643.863}
SPL {X  -155.811, Y  +731.738, Z    +0.000, E1   -70.890, E3 +142652.871}
SPL {X  -152.643, Y  +739.844, Z    +0.000, E1   -70.463, E3 +142661.730}
SPL {X  -149.782, Y  +746.247, Z    +0.000, E1   -70.149, E3 +142668.420}
SPL {X  -146.450, Y  +752.910, Z    +0.000, E1   -69.680, E3 +142676.298}
SPL {X  -143.017, Y  +759.082, Z    +0.000, E1   -69.156, E3 +142683.909}
SPL {X  -139.030, Y  +765.558, Z    +0.000, E1   -68.719, E3 +142690.942}
SPL {X  -134.589, Y  +772.070, Z    +0.000, E1   -68.090, E3 +142698.792}
SPL {X  -129.830, Y  +778.379, Z    +0.000, E1   -67.491, E3 +142705.801}
SPL {X  -116.788, Y  +792.975, Z    +0.000, E1   -71.297, E3 +142699.185}
SPL {X   -64.927, Y  +827.895, Z    +0.000, E1   -57.691, E3 +142824.788}
ENDSPLINE

SPLINE
SPL {X  -111.648, Y  +797.871, Z    +0.000, E1   -60.847, E3 +143021.771}
SPL {X  -149.288, Y  +747.285, Z    +0.000, E1   -46.770, E3 +143017.762}
SPL {X  -161.496, Y  +712.364, Z    +0.000, E1   -31.137, E3 +143023.557}
SPL {X  -164.701, Y  +693.202, Z    +0.000, E1   -17.512, E3 +143022.531}
SPL {X  -165.453, Y  +683.578, Z    +0.000, E1    -9.445, E3 +143021.733}
SPL {X  -165.642, Y  +677.105, Z    +0.000, E1    -3.559, E3 +143022.043}
SPL {X  -165.650, Y  +673.263, Z    +0.000, E1    +0.216, E3 +143020.803}
SPL {X  -165.650, Y  +670.095, Z    +0.000, E1    +6.482, E3 +143020.207}
SPL {X  -165.650, Y  +666.485, Z    +0.000, E1   +14.169, E3 +143020.106}
SPL {X  -165.650, Y  +661.236, Z    +0.000, E1   +26.072, E3 +143019.795}
SPL {X  -165.650, Y  +653.063, Z    +0.000, E1   +42.395, E3 +143019.199}
SPL {X  -165.650, Y  +640.535, Z    +0.000, E1   +60.776, E3 +143016.684}
SPL {X  -165.650, Y  +618.963, Z    +0.000, E1   +72.815, E3 +143016.663}
SPL {X  -165.650, Y  +575.208, Z    +0.000, E1   +76.222, E3 +143027.924}
SPL {X  -165.650, Y  +394.754, Z    +0.000, E1   +73.248, E3 +143123.070}
ENDSPLINE

SPLINE
SPL {X  -165.650, Y  +407.500, Z    +0.000, E1   +70.919, E3 +143137.691}
ENDSPLINE

SPLINE
SPL {X  -165.650, Y  +390.855, Z    +0.000, E1   +71.004, E3 +143148.619}
SPL {X  -165.534, Y  +372.295, Z    +0.000, E1   +71.066, E3 +143161.169}
SPL {X  -164.687, Y  +360.663, Z    +0.000, E1   +70.826, E3 +143171.461}
SPL {X  -162.841, Y  +348.123, Z    +0.000, E1   +70.683, E3 +143181.840}
SPL {X  -162.352, Y  +345.609, Z    +0.000, E1   +69.290, E3 +143195.793}
SPL {X  -157.663, Y  +327.685, Z    +0.000, E1   +69.808, E3 +143204.653}
SPL {X  -152.892, Y  +314.750, Z    +0.000, E1   +69.675, E3 +143214.869}
SPL {X  -149.246, Y  +306.628, Z    +0.000, E1   +69.029, E3 +143225.337}
SPL {X  -145.495, Y  +299.310, Z    +0.000, E1   +68.659, E3 +143232.946}
SPL {X  -141.249, Y  +291.963, Z    +0.000, E1   +68.223, E3 +143240.926}
SPL {X  -137.649, Y  +286.345, Z    +0.000, E1   +67.498, E3 +143248.862}
SPL {X  -134.450, Y  +281.737, Z    +0.000, E1   +67.268, E3 +143253.252}
SPL {X  -131.812, Y  +278.173, Z    +0.000, E1   +66.669, E3 +143258.601}
SPL {X  -128.148, Y  +273.533, Z    +0.000, E1   +67.328, E3 +143258.959}
SPL {X  -116.216, Y  +260.459, Z    +0.000, E1   +70.200, E3 +143255.266}
SPL {X   -66.125, Y  +226.621, Z    +0.000, E1   +55.862, E3 +143418.164}
ENDSPLINE

SPLINE
SPL {X  -111.531, Y  +256.023, Z    +0.000, E1   +58.853, E3 +143561.046}
SPL {X  -139.240, Y  +288.767, Z    +0.000, E1   +52.898, E3 +143571.219}
SPL {X  -156.827, Y  +325.161, Z    +0.000, E1   +39.042, E3 +143569.588}
SPL {X  -163.133, Y  +349.734, Z    +0.000, E1   +25.193, E3 +143570.713}
SPL {X  -165.214, Y  +366.494, Z    +0.000, E1   +12.605, E3 +143570.186}
SPL {X  -165.646, Y  +377.353, Z    +0.000, E1    +3.112, E3 +143569.452}
SPL {X  -165.650, Y  +380.500, Z    +0.000, E1    -0.000, E3 +143568.578}
SPL {X  -165.650, Y  +381.828, Z    +0.000, E1    -2.219, E3 +143568.030}
SPL {X  -165.650, Y  +385.044, Z    +0.000, E1    -8.496, E3 +143567.830}
SPL {X  -165.650, Y  +388.717, Z    +0.000, E1   -16.400, E3 +143567.685}
SPL {X  -165.650, Y  +394.613, Z    +0.000, E1   -29.184, E3 +143567.154}
SPL {X  -165.650, Y  +402.836, Z    +0.000, E1   -44.797, E3 +143566.557}
SPL {X  -165.650, Y  +416.111, Z    +0.000, E1   -60.729, E3 +143565.623}
SPL {X  -165.650, Y  +457.077, Z    +0.000, E1   -75.210, E3 +143568.947}
SPL {X  -165.650, Y  +475.293, Z    +0.000, E1   -75.741, E3 +143574.725}
SPL {X  -164.204, Y  +697.342, Z    +0.000, E1   -76.015, E3 +143661.699}
ENDSPLINE

SPLINE
SPL {X  -165.650, Y  +664.340, Z    +0.000, E1   -71.862, E3 +143687.103}
ENDSPLINE

SPLINE
SPL {X  -165.116, Y  +688.792, Z    +0.000, E1   -71.759, E3 +143704.543}
SPL {X  -162.089, Y  +709.665, Z    +0.000, E1   -71.739, E3 +143718.596}
SPL {X  -159.776, Y  +719.221, Z    +0.000, E1   -71.038, E3 +143731.418}
SPL {X  -155.811, Y  +731.738, Z    +0.000, E1   -70.890, E3 +143741.106}
SPL {X  -152.643, Y  +739.844, Z    +0.000, E1   -70.463, E3 +143749.966}
SPL {X  -149.782, Y  +746.247, Z    +0.000, E1   -70.149, E3 +143756.655}
SPL {X  -146.450, Y  +752.910, Z    +0.000, E1   -69.680, E3 +143764.534}
SPL {X  -143.017, Y  +759.082, Z    +0.000, E1   -69.156, E3 +143772.145}
SPL {X  -139.030, Y  +765.558, Z    +0.000, E1   -68.719, E3 +143779.178}
SPL {X  -134.589, Y  +772.070, Z    +0.000, E1   -68.090, E3 +143787.027}
SPL {X  -129.830, Y  +778.379, Z    +0.000, E1   -67.491, E3 +143794.037}
SPL {X  -116.788, Y  +792.975, Z    +0.000, E1   -71.297, E3 +143787.421}
SPL {X   -64.927, Y  +827.895, Z    +0.000, E1   -57.691, E3 +143913.024}
ENDSPLINE

SPLINE
SPL {X  -111.648, Y  +797.871, Z    +0.000, E1   -60.847, E3 +144110.006}
SPL {X  -149.288, Y  +747.285, Z    +0.000, E1   -46.770, E3 +144105.997}
SPL {X  -159.627, Y  +719.761, Z    +0.000, E1   -35.247, E3 +144111.062}
SPL {X  -164.185, Y  +697.485, Z    +0.000, E1   -20.950, E3 +144111.381}
SPL {X  -165.594, Y  +679.817, Z    +0.000, E1    -6.204, E3 +144110.157}
SPL {X  -165.650, Y  +673.522, Z    +0.000, E1    -0.038, E3 +144109.126}
SPL {X  -165.650, Y  +671.354, Z    +0.000, E1    +3.728, E3 +144108.614}
SPL {X  -165.650, Y  +666.485, Z    +0.000, E1   +14.169, E3 +144108.341}
SPL {X  -165.650, Y  +661.236, Z    +0.000, E1   +26.072, E3 +144108.030}
SPL {X  -165.650, Y  +653.063, Z    +0.000, E1   +42.395, E3 +144107.434}
SPL {X  -165.650, Y  +640.535, Z    +0.000, E1   +60.776, E3 +144104.919}
SPL {X  -165.650, Y  +618.963, Z    +0.000, E1   +72.815, E3 +144104.898}
SPL {X  -165.650, Y  +582.897, Z    +0.000, E1   +76.147, E3 +144113.559}
SPL {X  -165.650, Y  +558.388, Z    +0.000, E1   +76.294, E3 +144121.872}
SPL {X  -165.650, Y  +391.690, Z    +0.000, E1   +75.504, E3 +144191.638}
ENDSPLINE

SPLINE
SPL {X  -165.650, Y  +396.283, Z    +0.000, E1   +72.775, E3 +144214.943}
SPL {X  -165.650, Y  +407.500, Z    +0.000, E1   +70.919, E3 +144225.927}
ENDSPLINE

SPLINE
SPL {X  -165.650, Y  +384.687, Z    +0.000, E1   +71.028, E3 +144241.172}
SPL {X  -164.996, Y  +363.797, Z    +0.000, E1   +70.987, E3 +144256.147}
SPL {X  -162.841, Y  +348.123, Z    +0.000, E1   +70.683, E3 +144270.075}
SPL {X  -162.352, Y  +345.609, Z    +0.000, E1   +69.290, E3 +144284.028}
SPL {X  -157.663, Y  +327.685, Z    +0.000, E1   +69.808, E3 +144292.889}
SPL {X  -152.892, Y  +314.750, Z    +0.000, E1   +69.675, E3 +144303.104}
SPL {X  -149.246, Y  +306.628, Z    +0.000, E1   +69.029, E3 +144313.572}
SPL {X  -144.614, Y  +297.712, Z    +0.000, E1   +68.717, E3 +144321.926}
SPL {X  -141.011, Y  +291.576, Z    +0.000, E1   +68.040, E3 +144330.404}
SPL {X  -137.649, Y  +286.345, Z    +0.000, E1   +67.498, E3 +144337.097}
SPL {X  -134.450, Y  +281.737, Z    +0.000, E1   +67.268, E3 +144341.488}
SPL {X  -131.812, Y  +278.173, Z    +0.000, E1   +66.669, E3 +144346.836}
SPL {X  -128.148, Y  +273.533, Z    +0.000, E1   +67.328, E3 +144347.194}
SPL {X  -116.216, Y  +260.459, Z    +0.000, E1   +70.200, E3 +144343.501}
SPL {X   -66.125, Y  +226.621, Z    +0.000, E1   +55.862, E3 +144506.399}
ENDSPLINE

SPLINE
SPL {X  -111.531, Y  +256.023, Z    +0.000, E1   +58.853, E3 +144649.281}
SPL {X  -139.240, Y  +288.767, Z    +0.000, E1   +52.898, E3 +144659.454}
SPL {X  -156.827, Y  +325.161, Z    +0.000, E1   +39.042, E3 +144657.823}
SPL {X  -162.324, Y  +345.471, Z    +0.000, E1   +27.849, E3 +144658.292}
SPL {X  -165.055, Y  +364.477, Z    +0.000, E1   +14.326, E3 +144658.730}
SPL {X  -165.646, Y  +377.353, Z    +0.000, E1    +3.112, E3 +144657.687}
SPL {X  -165.650, Y  +380.500, Z    +0.000, E1    -0.000, E3 +144656.813}
SPL {X  -165.650, Y  +381.828, Z    +0.000, E1    -2.219, E3 +144656.265}
SPL {X  -165.650, Y  +385.044, Z    +0.000, E1    -8.496, E3 +144656.065}
SPL {X  -165.650, Y  +388.717, Z    +0.000, E1   -16.400, E3 +144655.921}
SPL {X  -165.650, Y  +394.613, Z    +0.000, E1   -29.184, E3 +144655.390}
SPL {X  -165.650, Y  +402.836, Z    +0.000, E1   -44.797, E3 +144654.792}
SPL {X  -165.650, Y  +416.111, Z    +0.000, E1   -60.729, E3 +144653.859}
SPL {X  -165.650, Y  +471.994, Z    +0.000, E1   -75.670, E3 +144661.912}
SPL {X  -164.204, Y  +697.342, Z    +0.000, E1   -76.015, E3 +144749.935}
ENDSPLINE

SPLINE
SPL {X  -165.650, Y  +656.030, Z    +0.000, E1   -71.686, E3 +144771.374}
ENDSPLINE

SPLINE
SPL {X  -165.610, Y  +679.119, Z    +0.000, E1   -71.889, E3 +144784.997}
SPL {X  -164.561, Y  +694.465, Z    +0.000, E1   -71.736, E3 +144796.631}
SPL {X  -162.089, Y  +709.665, Z    +0.000, E1   -71.739, E3 +144806.831}
SPL {X  -159.776, Y  +719.221, Z    +0.000, E1   -71.038, E3 +144819.654}
SPL {X  -155.811, Y  +731.738, Z    +0.000, E1   -70.890, E3 +144829.342}
SPL {X  -152.643, Y  +739.844, Z    +0.000, E1   -70.463, E3 +144838.201}
SPL {X  -149.782, Y  +746.247, Z    +0.000, E1   -70.149, E3 +144844.891}
SPL {X  -146.450, Y  +752.910, Z    +0.000, E1   -69.680, E3 +144852.769}
SPL {X  -143.017, Y  +759.082, Z    +0.000, E1   -69.156, E3 +144860.380}
SPL {X  -140.057, Y  +763.953, Z    +0.000, E1   -68.829, E3 +144865.619}
SPL {X  -136.535, Y  +769.298, Z    +0.000, E1   -68.442, E3 +144871.481}
SPL {X  -133.553, Y  +773.498, Z    +0.000, E1   -67.773, E3 +144877.646}
SPL {X  -129.830, Y  +778.379, Z    +0.000, E1   -67.491, E3 +144882.272}
SPL {X  -116.788, Y  +792.975, Z    +0.000, E1   -71.297, E3 +144875.656}
SPL {X   -64.927, Y  +827.895, Z    +0.000, E1   -57.691, E3 +145001.259}
ENDSPLINE

SPLINE
SPL {X  -111.648, Y  +797.871, Z    +0.000, E1   -60.847, E3 +145198.241}
SPL {X  -149.288, Y  +747.285, Z    +0.000, E1   -46.770, E3 +145194.232}
SPL {X  -159.627, Y  +719.761, Z    +0.000, E1   -35.247, E3 +145199.297}
SPL {X  -164.185, Y  +697.485, Z    +0.000, E1   -20.950, E3 +145199.616}
SPL {X  -165.594, Y  +679.817, Z    +0.000, E1    -6.204, E3 +145198.393}
SPL {X  -165.650, Y  +673.522, Z    +0.000, E1    -0.038, E3 +145197.362}
SPL {X  -165.650, Y  +671.354, Z    +0.000, E1    +3.728, E3 +145196.849}
SPL {X  -165.650, Y  +666.485, Z    +0.000, E1   +14.169, E3 +145196.576}
SPL {X  -165.650, Y  +661.236, Z    +0.000, E1   +26.072, E3 +145196.266}
SPL {X  -165.650, Y  +653.063, Z    +0.000, E1   +42.395, E3 +145195.670}
SPL {X  -165.650, Y  +640.535, Z    +0.000, E1   +60.776, E3 +145193.154}
SPL {X  -165.650, Y  +618.963, Z    +0.000, E1   +72.815, E3 +145193.133}
SPL {X  -165.650, Y  +582.897, Z    +0.000, E1   +76.147, E3 +145201.795}
SPL {X  -165.650, Y  +558.388, Z    +0.000, E1   +76.294, E3 +145210.107}
SPL {X  -165.650, Y  +391.690, Z    +0.000, E1   +75.504, E3 +145279.873}
ENDSPLINE

SPLINE
SPL {X  -165.650, Y  +396.283, Z    +0.000, E1   +72.775, E3 +145303.178}
SPL {X  -165.650, Y  +407.500, Z    +0.000, E1   +70.919, E3 +145314.162}
ENDSPLINE

SPLINE
SPL {X  -165.650, Y  +384.687, Z    +0.000, E1   +71.028, E3 +145329.408}
SPL {X  -164.996, Y  +363.797, Z    +0.000, E1   +70.987, E3 +145344.383}
SPL {X  -162.841, Y  +348.123, Z    +0.000, E1   +70.683, E3 +145358.311}
SPL {X  -162.352, Y  +345.609, Z    +0.000, E1   +69.290, E3 +145372.264}
SPL {X  -157.663, Y  +327.685, Z    +0.000, E1   +69.808, E3 +145381.124}
ENDSPLINE

SPLINE
SPL {X  -158.659, Y  +330.884, Z    +0.000, E1   +67.335, E3 +145398.346}
ENDSPLINE

SPLINE
SPL {X  -155.058, Y  +320.218, Z    +0.000, E1   +66.982, E3 +145409.597}
SPL {X  -151.047, Y  +310.495, Z    +0.000, E1   +66.593, E3 +145420.231}
SPL {X  -146.639, Y  +301.448, Z    +0.000, E1   +65.839, E3 +145432.440}
SPL {X  -142.469, Y  +293.987, Z    +0.000, E1   +65.133, E3 +145442.489}
SPL {X  -139.022, Y  +288.429, Z    +0.000, E1   +64.807, E3 +145448.687}
SPL {X  -136.717, Y  +284.968, Z    +0.000, E1   +64.044, E3 +145455.280}
SPL {X  -133.061, Y  +279.835, Z    +0.000, E1   +64.204, E3 +145458.693}
SPL {X  -118.927, Y  +263.191, Z    +0.000, E1   +67.951, E3 +145454.706}
SPL {X   -76.819, Y  +231.739, Z    +0.000, E1   +54.834, E3 +145632.712}
ENDSPLINE

SPLINE
SPL {X  -140.879, Y  +291.363, Z    +0.000, E1   +48.273, E3 +145740.153}
SPL {X  -158.845, Y  +331.507, Z    +0.000, E1   +33.834, E3 +145749.488}
SPL {X  -164.164, Y  +356.358, Z    +0.000, E1   +18.707, E3 +145745.810}
SPL {X  -165.341, Y  +368.384, Z    +0.000, E1   +10.076, E3 +145746.555}
SPL {X  -165.648, Y  +377.641, Z    +0.000, E1    +2.653, E3 +145745.905}
SPL {X  -165.650, Y  +380.500, Z    +0.000, E1    -0.000, E3 +145744.936}
SPL {X  -165.650, Y  +381.694, Z    +0.000, E1    -1.679, E3 +145744.338}
SPL {X  -165.650, Y  +385.900, Z    +0.000, E1    -8.711, E3 +145744.160}
SPL {X  -165.650, Y  +390.854, Z    +0.000, E1   -18.692, E3 +145743.336}
SPL {X  -165.650, Y  +395.801, Z    +0.000, E1   -28.236, E3 +145743.335}
SPL {X  -165.650, Y  +403.802, Z    +0.000, E1   -41.748, E3 +145743.156}
SPL {X  -165.650, Y  +418.088, Z    +0.000, E1   -59.974, E3 +145740.429}
SPL {X  -165.650, Y  +461.994, Z    +0.000, E1   -72.657, E3 +145748.566}
SPL {X  -165.650, Y  +492.072, Z    +0.000, E1   -73.925, E3 +145758.669}
SPL {X  -165.650, Y  +640.142, Z    +0.000, E1   -72.635, E3 +145837.545}
ENDSPLINE

SPLINE
SPL {X  -165.650, Y  +619.423, Z    +0.000, E1   -68.618, E3 +145859.742}
ENDSPLINE

SPLINE
SPL {X  -165.650, Y  +635.985, Z    +0.000, E1   -68.274, E3 +145875.945}
SPL {X  -165.650, Y  +647.687, Z    +0.000, E1   -68.151, E3 +145886.445}
SPL {X  -165.650, Y  +665.917, Z    +0.000, E1   -68.414, E3 +145899.205}
SPL {X  -165.417, Y  +684.287, Z    +0.000, E1   -68.467, E3 +145913.502}
SPL {X  -164.268, Y  +696.853, Z    +0.000, E1   -68.071, E3 +145927.131}
SPL {X  -161.478, Y  +712.444, Z    +0.000, E1   -67.895, E3 +145941.338}
SPL {X  -157.774, Y  +725.970, Z    +0.000, E1   -67.383, E3 +145956.340}
SPL {X  -154.751, Y  +734.593, Z    +0.000, E1   -66.864, E3 +145966.934}
SPL {X  -151.443, Y  +742.618, Z    +0.000, E1   -66.527, E3 +145975.929}
SPL {X  -148.198, Y  +749.508, Z    +0.000, E1   -66.065, E3 +145984.410}
SPL {X  -144.642, Y  +756.238, Z    +0.000, E1   -65.678, E3 +145992.276}
SPL {X  -140.398, Y  +763.411, Z    +0.000, E1   -64.853, E3 +146002.753}
SPL {X  -135.180, Y  +771.240, Z    +0.000, E1   -64.104, E3 +146012.802}
SPL {X  -125.028, Y  +784.164, Z    +0.000, E1   -66.760, E3 +146011.272}
SPL {X   -71.589, Y  +824.882, Z    +0.000, E1   -56.415, E3 +146138.337}
ENDSPLINE

SPLINE
SPL {X  -127.072, Y  +781.767, Z    +0.000, E1   -54.186, E3 +146301.309}
SPL {X  -150.680, Y  +744.314, Z    +0.000, E1   -44.608, E3 +146312.265}
SPL {X  -162.376, Y  +708.273, Z    +0.000, E1   -25.870, E3 +146304.389}
SPL {X  -165.092, Y  +689.091, Z    +0.000, E1   -12.938, E3 +146305.808}
SPL {X  -165.629, Y  +678.122, Z    +0.000, E1    -4.178, E3 +146304.955}
SPL {X  -165.650, Y  +673.539, Z    +0.000, E1    -0.057, E3 +146304.053}
SPL {X  -165.650, Y  +671.359, Z    +0.000, E1    +3.116, E3 +146303.410}
SPL {X  -165.650, Y  +667.465, Z    +0.000, E1   +10.413, E3 +146303.204}
SPL {X  -165.650, Y  +662.220, Z    +0.000, E1   +20.600, E3 +146302.896}
SPL {X  -165.650, Y  +652.464, Z    +0.000, E1   +39.379, E3 +146301.843}
SPL {X  -165.650, Y  +636.657, Z    +0.000, E1   +60.410, E3 +146299.132}
SPL {X  -165.650, Y  +613.310, Z    +0.000, E1   +72.038, E3 +146299.491}
SPL {X  -165.650, Y  +568.914, Z    +0.000, E1   +74.438, E3 +146314.076}
SPL {X  -165.650, Y  +420.321, Z    +0.000, E1   +71.570, E3 +146402.729}
ENDSPLINE

SPLINE
SPL {X  -165.650, Y  +437.633, Z    +0.000, E1   +68.421, E3 +146418.477}
ENDSPLINE

SPLINE
SPL {X  -164.513, Y  +359.128, Z    +0.000, E1   +73.170, E3 +146428.711}
SPL {X  -163.967, Y  +354.944, Z    +0.000, E1   +72.327, E3 +146440.064}
SPL {X  -163.372, Y  +351.124, Z    +0.000, E1   +71.295, E3 +146452.656}
SPL {X  -162.653, Y  +347.134, Z    +0.000, E1   +70.371, E3 +146463.892}
SPL {X  -161.430, Y  +341.349, Z    +0.000, E1   +69.492, E3 +146475.966}
SPL {X  -160.389, Y  +337.084, Z    +0.000, E1   +68.301, E3 +146489.053}
SPL {X  -159.245, Y  +332.881, Z    +0.000, E1   +67.496, E3 +146498.713}
SPL {X  -157.072, Y  +325.885, Z    +0.000, E1   +67.020, E3 +146508.062}
SPL {X  -154.432, Y  +318.577, Z    +0.000, E1   +66.843, E3 +146515.267}
SPL {X  -151.047, Y  +310.495, Z    +0.000, E1   +66.593, E3 +146523.679}
SPL {X  -146.639, Y  +301.448, Z    +0.000, E1   +65.839, E3 +146535.889}
SPL {X  -142.469, Y  +293.987, Z    +0.000, E1   +65.133, E3 +146545.937}
SPL {X  -139.022, Y  +288.429, Z    +0.000, E1   +64.807, E3 +146552.136}
SPL {X  -136.717, Y  +284.968, Z    +0.000, E1   +64.044, E3 +146558.728}
SPL {X  -133.061, Y  +279.835, Z    +0.000, E1   +64.204, E3 +146562.142}
SPL {X  -118.927, Y  +263.191, Z    +0.000, E1   +67.951, E3 +146558.154}
SPL {X   -76.819, Y  +231.739, Z    +0.000, E1   +54.834, E3 +146736.160}
ENDSPLINE

SPLINE
SPL {X  -140.879, Y  +291.363, Z    +0.000, E1   +48.273, E3 +146843.601}
SPL {X  -158.845, Y  +331.507, Z    +0.000, E1   +33.834, E3 +146852.936}
SPL {X  -164.164, Y  +356.358, Z    +0.000, E1   +18.707, E3 +146849.259}
SPL {X  -165.341, Y  +368.384, Z    +0.000, E1   +10.076, E3 +146850.003}
SPL {X  -165.648, Y  +377.641, Z    +0.000, E1    +2.653, E3 +146849.354}
SPL {X  -165.650, Y  +380.500, Z    +0.000, E1    -0.000, E3 +146848.384}
SPL {X  -165.650, Y  +381.694, Z    +0.000, E1    -1.679, E3 +146847.786}
SPL {X  -165.650, Y  +384.595, Z    +0.000, E1    -6.546, E3 +146847.648}
SPL {X  -165.650, Y  +389.276, Z    +0.000, E1   -15.245, E3 +146847.156}
SPL {X  -165.650, Y  +395.801, Z    +0.000, E1   -28.236, E3 +146846.783}
SPL {X  -165.650, Y  +403.802, Z    +0.000, E1   -41.748, E3 +146846.604}
SPL {X  -165.650, Y  +419.045, Z    +0.000, E1   -60.641, E3 +146843.925}
SPL {X  -165.650, Y  +474.102, Z    +0.000, E1   -73.446, E3 +146855.709}
SPL {X  -165.650, Y  +640.142, Z    +0.000, E1   -72.635, E3 +146940.993}
ENDSPLINE

SPLINE
SPL {X  -165.650, Y  +612.217, Z    +0.000, E1   -68.647, E3 +146956.919}
ENDSPLINE

SPLINE
SPL {X  -165.650, Y  +623.643, Z    +0.000, E1   -68.543, E3 +146967.015}
SPL {X  -165.650, Y  +635.985, Z    +0.000, E1   -68.274, E3 +146979.394}
SPL {X  -165.650, Y  +656.072, Z    +0.000, E1   -68.403, E3 +146994.688}
SPL {X  -165.650, Y  +673.246, Z    +0.000, E1   -68.189, E3 +147010.443}
SPL {X  -164.760, Y  +692.647, Z    +0.000, E1   -68.400, E3 +147024.409}
SPL {X  -162.986, Y  +705.089, Z    +0.000, E1   -67.915, E3 +147038.620}
SPL {X  -159.812, Y  +719.091, Z    +0.000, E1   -67.711, E3 +147051.619}
SPL {X  -156.969, Y  +728.420, Z    +0.000, E1   -67.278, E3 +147062.401}
SPL {X  -153.458, Y  +737.875, Z    +0.000, E1   -66.902, E3 +147072.863}
SPL {X  -149.433, Y  +746.982, Z    +0.000, E1   -66.131, E3 +147085.494}
SPL {X  -144.642, Y  +756.238, Z    +0.000, E1   -65.678, E3 +147095.725}
SPL {X  -140.398, Y  +763.411, Z    +0.000, E1   -64.853, E3 +147106.201}
SPL {X  -135.180, Y  +771.240, Z    +0.000, E1   -64.104, E3 +147116.250}
SPL {X  -125.028, Y  +784.164, Z    +0.000, E1   -66.760, E3 +147114.720}
SPL {X   -71.589, Y  +824.882, Z    +0.000, E1   -56.415, E3 +147241.785}
ENDSPLINE

SPLINE
SPL {X  -127.072, Y  +781.767, Z    +0.000, E1   -54.186, E3 +147404.757}
SPL {X  -150.680, Y  +744.314, Z    +0.000, E1   -44.608, E3 +147415.714}
SPL {X  -162.376, Y  +708.273, Z    +0.000, E1   -25.870, E3 +147407.837}
SPL {X  -165.092, Y  +689.091, Z    +0.000, E1   -12.938, E3 +147409.256}
SPL {X  -165.629, Y  +678.122, Z    +0.000, E1    -4.178, E3 +147408.403}
SPL {X  -165.650, Y  +673.539, Z    +0.000, E1    -0.057, E3 +147407.501}
SPL {X  -165.650, Y  +671.359, Z    +0.000, E1    +3.116, E3 +147406.858}
SPL {X  -165.650, Y  +665.277, Z    +0.000, E1   +14.409, E3 +147406.503}
SPL {X  -165.650, Y  +659.573, Z    +0.000, E1   +26.182, E3 +147406.251}
SPL {X  -165.650, Y  +652.464, Z    +0.000, E1   +39.379, E3 +147405.292}
SPL {X  -165.650, Y  +634.871, Z    +0.000, E1   +61.762, E3 +147402.524}
SPL {X  -165.650, Y  +574.769, Z    +0.000, E1   +74.441, E3 +147415.172}
SPL {X  -165.650, Y  +420.321, Z    +0.000, E1   +71.570, E3 +147506.177}
ENDSPLINE

SPLINE
SPL {X  -165.650, Y  +437.633, Z    +0.000, E1   +68.421, E3 +147521.926}
ENDSPLINE

SPLINE
SPL {X  -164.513, Y  +359.128, Z    +0.000, E1   +73.170, E3 +147532.159}
SPL {X  -163.967, Y  +354.944, Z    +0.000, E1   +72.327, E3 +147543.512}
SPL {X  -163.571, Y  +352.336, Z    +0.000, E1   +71.524, E3 +147552.930}
SPL {X  -162.836, Y  +348.099, Z    +0.000, E1   +70.646, E3 +147564.404}
SPL {X  -161.430, Y  +341.349, Z    +0.000, E1   +69.492, E3 +147579.414}
SPL {X  -160.389, Y  +337.084, Z    +0.000, E1   +68.301, E3 +147592.502}
SPL {X  -158.795, Y  +331.340, Z    +0.000, E1   +67.291, E3 +147605.188}
SPL {X  -154.229, Y  +318.056, Z    +0.000, E1   +66.925, E3 +147618.792}
SPL {X  -149.308, Y  +306.758, Z    +0.000, E1   +66.321, E3 +147631.998}
SPL {X  -145.703, Y  +299.692, Z    +0.000, E1   +65.663, E3 +147641.673}
SPL {X  -142.469, Y  +293.987, Z    +0.000, E1   +65.133, E3 +147649.385}
SPL {X  -139.022, Y  +288.429, Z    +0.000, E1   +64.807, E3 +147655.584}
SPL {X  -136.717, Y  +284.968, Z    +0.000, E1   +64.044, E3 +147662.176}
SPL {X  -133.061, Y  +279.835, Z    +0.000, E1   +64.204, E3 +147665.590}
SPL {X  -118.927, Y  +263.191, Z    +0.000, E1   +67.951, E3 +147661.602}
SPL {X   -76.819, Y  +231.739, Z    +0.000, E1   +54.834, E3 +147839.608}
ENDSPLINE

SPLINE
SPL {X  -140.879, Y  +291.363, Z    +0.000, E1   +48.273, E3 +147947.050}
SPL {X  -158.845, Y  +331.507, Z    +0.000, E1   +33.834, E3 +147956.384}
SPL {X  -164.164, Y  +356.358, Z    +0.000, E1   +18.707, E3 +147952.707}
SPL {X  -165.341, Y  +368.384, Z    +0.000, E1   +10.076, E3 +147953.451}
SPL {X  -165.648, Y  +377.641, Z    +0.000, E1    +2.653, E3 +147952.802}
SPL {X  -165.650, Y  +380.939, Z    +0.000, E1    -0.407, E3 +147951.613}
SPL {X  -165.650, Y  +384.595, Z    +0.000, E1    -6.546, E3 +147951.096}
SPL {X  -165.650, Y  +389.276, Z    +0.000, E1   -15.245, E3 +147950.604}
SPL {X  -165.650, Y  +395.801, Z    +0.000, E1   -28.236, E3 +147950.232}
SPL {X  -165.650, Y  +403.802, Z    +0.000, E1   -41.748, E3 +147950.053}
SPL {X  -165.650, Y  +418.088, Z    +0.000, E1   -59.974, E3 +147947.325}
SPL {X  -165.650, Y  +461.994, Z    +0.000, E1   -72.657, E3 +147955.463}
SPL {X  -165.650, Y  +492.072, Z    +0.000, E1   -73.925, E3 +147965.565}
SPL {X  -165.650, Y  +637.039, Z    +0.000, E1   -73.842, E3 +148032.230}
ENDSPLINE

SPLINE
SPL {X  -165.650, Y  +617.598, Z    +0.000, E1   -69.273, E3 +148059.297}
ENDSPLINE

SPLINE
SPL {X  -165.650, Y  +623.643, Z    +0.000, E1   -68.543, E3 +148070.463}
SPL {X  -165.650, Y  +635.985, Z    +0.000, E1   -68.274, E3 +148082.842}
SPL {X  -165.650, Y  +647.687, Z    +0.000, E1   -68.151, E3 +148093.342}
SPL {X  -165.650, Y  +665.917, Z    +0.000, E1   -68.414, E3 +148106.101}
SPL {X  -165.417, Y  +684.287, Z    +0.000, E1   -68.467, E3 +148120.398}
SPL {X  -164.268, Y  +696.853, Z    +0.000, E1   -68.071, E3 +148134.028}
SPL {X  -162.443, Y  +707.938, Z    +0.000, E1   -67.853, E3 +148144.762}
SPL {X  -159.812, Y  +719.091, Z    +0.000, E1   -67.711, E3 +148155.068}
SPL {X  -156.969, Y  +728.420, Z    +0.000, E1   -67.278, E3 +148165.850}
SPL {X  -154.751, Y  +734.593, Z    +0.000, E1   -66.864, E3 +148173.831}
SPL {X  -151.443, Y  +742.618, Z    +0.000, E1   -66.527, E3 +148182.826}
SPL {X  -148.198, Y  +749.508, Z    +0.000, E1   -66.065, E3 +148191.307}
SPL {X  -144.642, Y  +756.238, Z    +0.000, E1   -65.678, E3 +148199.173}
SPL {X  -140.398, Y  +763.411, Z    +0.000, E1   -64.853, E3 +148209.649}
SPL {X  -135.180, Y  +771.240, Z    +0.000, E1   -64.104, E3 +148219.699}
SPL {X  -125.028, Y  +784.164, Z    +0.000, E1   -66.760, E3 +148218.168}
SPL {X   -74.840, Y  +823.280, Z    +0.000, E1   -57.857, E3 +148318.701}
SPL {X   -70.065, Y  +825.603, Z    +0.000, E1   -55.379, E3 +148379.003}
ENDSPLINE

SPLINE
SPL {X  -127.072, Y  +781.767, Z    +0.000, E1   -54.186, E3 +148508.206}
SPL {X  -150.680, Y  +744.314, Z    +0.000, E1   -44.608, E3 +148519.162}
SPL {X  -162.376, Y  +708.273, Z    +0.000, E1   -25.870, E3 +148511.286}
SPL {X  -165.092, Y  +689.091, Z    +0.000, E1   -12.938, E3 +148512.704}
SPL {X  -165.629, Y  +678.122, Z    +0.000, E1    -4.178, E3 +148511.852}
SPL {X  -165.650, Y  +673.539, Z    +0.000, E1    -0.057, E3 +148510.949}
SPL {X  -165.650, Y  +671.359, Z    +0.000, E1    +3.116, E3 +148510.306}
SPL {X  -165.650, Y  +665.277, Z    +0.000, E1   +14.409, E3 +148509.951}
SPL {X  -165.650, Y  +659.573, Z    +0.000, E1   +26.182, E3 +148509.699}
SPL {X  -165.650, Y  +652.464, Z    +0.000, E1   +39.379, E3 +148508.740}
SPL {X  -165.650, Y  +634.871, Z    +0.000, E1   +61.762, E3 +148505.973}
SPL {X  -165.650, Y  +574.769, Z    +0.000, E1   +74.441, E3 +148518.621}
SPL {X  -165.650, Y  +420.321, Z    +0.000, E1   +71.570, E3 +148609.626}
ENDSPLINE

SPLINE
SPL {X  -165.650, Y  +437.633, Z    +0.000, E1   +68.421, E3 +148625.374}
ENDSPLINE

SPLINE
SPL {X  -164.513, Y  +359.128, Z    +0.000, E1   +73.170, E3 +148635.607}
SPL {X  -163.967, Y  +354.944, Z    +0.000, E1   +72.327, E3 +148646.961}
SPL {X  -163.372, Y  +351.124, Z    +0.000, E1   +71.295, E3 +148659.553}
SPL {X  -162.653, Y  +347.134, Z    +0.000, E1   +70.371, E3 +148670.788}
SPL {X  -161.451, Y  +341.438, Z    +0.000, E1   +69.889, E3 +148679.107}
SPL {X  -161.444, Y  +341.410, Z    +0.000, E1   +69.001, E3 +148686.694}
SPL {X  -160.389, Y  +337.084, Z    +0.000, E1   +68.301, E3 +148695.950}
SPL {X  -158.795, Y  +331.340, Z    +0.000, E1   +67.291, E3 +148708.636}
SPL {X  -154.229, Y  +318.056, Z    +0.000, E1   +66.925, E3 +148722.240}
SPL {X  -149.308, Y  +306.758, Z    +0.000, E1   +66.321, E3 +148735.447}
SPL {X  -145.703, Y  +299.692, Z    +0.000, E1   +65.663, E3 +148745.121}
SPL {X  -142.469, Y  +293.987, Z    +0.000, E1   +65.133, E3 +148752.834}
SPL {X  -139.022, Y  +288.429, Z    +0.000, E1   +64.807, E3 +148759.032}
SPL {X  -136.717, Y  +284.968, Z    +0.000, E1   +64.044, E3 +148765.625}
SPL {X  -133.061, Y  +279.835, Z    +0.000, E1   +64.204, E3 +148769.038}
SPL {X  -118.927, Y  +263.191, Z    +0.000, E1   +67.951, E3 +148765.051}
SPL {X   -76.819, Y  +231.739, Z    +0.000, E1   +54.834, E3 +148943.057}
ENDSPLINE

SPLINE
SPL {X  -140.879, Y  +291.363, Z    +0.000, E1   +48.273, E3 +149050.498}
SPL {X  -158.845, Y  +331.507, Z    +0.000, E1   +33.834, E3 +149059.833}
SPL {X  -164.164, Y  +356.358, Z    +0.000, E1   +18.707, E3 +149056.155}
SPL {X  -165.519, Y  +371.910, Z    +0.000, E1    +7.409, E3 +149056.564}
SPL {X  -165.650, Y  +380.329, Z    +0.000, E1    +0.239, E3 +149055.410}
SPL {X  -165.650, Y  +381.694, Z    +0.000, E1    -1.679, E3 +149054.682}
SPL {X  -165.650, Y  +384.595, Z    +0.000, E1    -6.546, E3 +149054.544}
SPL {X  -165.650, Y  +389.276, Z    +0.000, E1   -15.245, E3 +149054.053}
SPL {X  -165.650, Y  +395.801, Z    +0.000, E1   -28.236, E3 +149053.680}
SPL {X  -165.650, Y  +403.802, Z    +0.000, E1   -41.748, E3 +149053.501}
SPL {X  -165.650, Y  +418.088, Z    +0.000, E1   -59.974, E3 +149050.773}
SPL {X  -165.650, Y  +461.994, Z    +0.000, E1   -72.657, E3 +149058.911}
SPL {X  -165.650, Y  +492.072, Z    +0.000, E1   -73.925, E3 +149069.013}
SPL {X  -165.650, Y  +640.142, Z    +0.000, E1   -72.635, E3 +149147.890}
ENDSPLINE

SPLINE
SPL {X  -165.650, Y  +619.423, Z    +0.000, E1   -68.618, E3 +149170.087}
ENDSPLINE

